# B&R Automation Studio project SD_SMA_SCADA_DEMO
Automation Studio 4.12.9.18 SP; technology packages: mapp 5.24.3, mappView 5.24.4

## Configuration Config1

CPU X20CP3687X, AutomationRuntime M4.93, Build 4.1.2, Safety 0.0, Vc V4.73.2

### Task classes (Cpu.sw)
```
Cyclic#4:
  AlarmQuerr <- AlarmQuerry.prg
  Trend <- Trend.prg
Binaries: udbdef, mvLoader, FWRules, TCData, arsvcreg, TCLang, sysconf, Role, User, iomap, ashwd, asfw, arconfig, ashwac, TC
Libraries: AsHttp, runtime, asstring, AsBrStr, sys_lib, LxVar, BrRand, MpAlarm, MpBase, arssl, fileio, astime, asieccon, brsystem, MpReport, standard
```

### Hardware
```
X20CP3687X : X20CP3687X v1.6.2.0
  Connector IF2:
    ActivateDevice = 1
    Mode = Manual
    InternetAddress = 192.168.50.233
    SubnetMask = 255.255.255.0
    InaPort = 0
    ActivateSnmp = 2
  ConfigurationID = SD_SMA_SCADA_DEMO_Config1
  UserPartitionSize = 100
  FileDevice1
  FileDeviceName1 = USER
  FileDevicePath1 = USER_PATH
  FtpUser1
  FtpUsername1 = br
  FtpUserPassword1 = JPl1VVziIj5tK4ypV/PCMk3zrwuEHr3/unO+8TvKNbo=  // 123
  FtpUserSalt1 = TmpN9Vd5
  FTPAccessRight1 = 0
  WebServerWebDir = D:\web\CFCARD\WEBROOT\
  WebServerStartPage = line.html
  ActivateOpcUa = 1
  OpcUaInformationModels_PV_Version = 1
```

## Configuration Config2

CPU X20CP3687X, AutomationRuntime M4.93, Build 4.1.2, Safety 0.0, Vc V4.73.2

### Task classes (Cpu.sw)
```
Cyclic#4:
  DataGen <- DataGen.prg
  DataRev <- DataRev.prg
  AlarmQuerr <- AlarmQuerry.prg [disabled]
  Trend <- Trend.prg [disabled]
Binaries: udbdef, mvLoader, FWRules, TCData, arsvcreg, TCLang, sysconf, Role, User, iomap, ashwd, asfw, arconfig, ashwac, TC
Libraries: AsHttp, runtime, asstring, AsBrStr, sys_lib, LxVar, BrRand, MpAlarm, MpBase, MpReport, arssl, fileio, astime, asieccon, brsystem
```

### Hardware
```
X20CP3687X : X20CP3687X v1.6.2.0
  Connector IF2:
    ActivateDevice = 1
    Mode = Manual
    InternetAddress = 192.168.50.233
    SubnetMask = 255.255.255.0
    InaPort = 0
    ActivateSnmp = 2
  ConfigurationID = SD_SMA_SCADA_DEMO_Config1
  UserPartitionSize = 100
  Simulation = 1
  FileDevice1
  FileDeviceName1 = USER
  FileDevicePath1 = USER_PATH
  FtpUser1
  FtpUsername1 = br
  FtpUserPassword1 = JPl1VVziIj5tK4ypV/PCMk3zrwuEHr3/unO+8TvKNbo=  // 123
  FtpUserSalt1 = TmpN9Vd5
  FTPAccessRight1 = 0
  WebServerWebDir = D:\web\CFCARD\WEBROOT\
  WebServerStartPage = line.html
  ActivateOpcUa = 1
  OpcUaInformationModels_PV_Version = 1
```

## Configuration PC3100

CPU X20CP1586, AutomationRuntime J4.93, Build 4.1.2, Safety 0.0, Vc V4.73.2

## Configuration cp1586

CPU 5APC3100.KBU2-000, AutomationRuntime J4.93, Build 4.1.2, Safety 0.0, Vc V4.73.2

### Task classes (Cpu.sw)
```
Cyclic#1:
  TimeSt <- TimeSt.prg
Cyclic#4:
  DataGen <- DataGen.prg
  DataRev <- DataRev.prg
  AlarmQuerr <- AlarmQuerry.prg
  Trend <- Trend.prg
  ParallelTe <- ParallelTest.prg
Binaries: udbdef, mvLoader, FWRules, TCData, arsvcreg, TCLang, sysconf, Role, User, iomap, ashwd, asfw, arconfig, ashwac, TC
Libraries: AsHttp, runtime, asstring, AsBrStr, sys_lib, LxVar, BrRand, MpAlarm, MpBase, MpReport, standard, arssl, fileio, astime, asieccon, brsystem
```

### Hardware
```
X20CP1586 : X20CP1586 v1.10.0.0
  Connector IF2:
    ActivateDevice = 1
    Mode = Manual
    InternetAddress = 192.168.50.233
    SubnetMask = 255.255.255.0
    InaPort = 0
    ActivateSnmp = 2
  Connector IF3:
    CycleTime = 400
  ConfigurationID = SD_SMA_SCADA_DEMO_Config1
  UserPartitionSize = 100
  FileDevice1
  FileDeviceName1 = USER
  FileDevicePath1 = USER_PATH
  FtpUser1
  FtpUsername1 = br
  FtpUserPassword1 = JPl1VVziIj5tK4ypV/PCMk3zrwuEHr3/unO+8TvKNbo=  // 123
  FtpUserSalt1 = TmpN9Vd5
  FTPAccessRight1 = 0
  WebServerWebDir = D:\web\CFCARD\WEBROOT\
  WebServerStartPage = line.html
  ActivateOpcUa = 1
  OpcUaInformationModels_PV_Version = 1
```

## Logical view

Binary libraries used (declarations not repeated): operator, runtime, astime, AsIecCon, AsHttp, asstring, AsBrStr, sys_lib, MpAlarm 5.24.3, MpBase, MpReport 5.24.3, standard

### Global.typ - Global data types
```iecst
TYPE
	dbReadConfig_typ : 	STRUCT
		strStartTime : ARRAY[0..DB_READ_QUERY_SIZE_MINUS_ONE]OF STRING[20];
		strEndTime : ARRAY[0..DB_READ_QUERY_SIZE_MINUS_ONE]OF STRING[20];
		strPointName : ARRAY[0..DB_READ_QUERY_SIZE_MINUS_ONE]OF STRING[20];
	END_STRUCT;
	dbReadRev_typ : 	STRUCT
		rRevBuffer : ARRAY[0..REV_BUFFER_SIZE_MINUS_ONE]OF REAL;
		udiRevTime : ARRAY[0..REV_BUFFER_SIZE_MINUS_ONE]OF UDINT;
		udiRevFeedBack : UDINT;
	END_STRUCT;
	dbReadQuery_typ : 	STRUCT
		stConfig : dbReadConfig_typ;
		stCmd : dbReadCmd_typ;
		stRev : ARRAY[0..DB_READ_QUERY_SIZE_MINUS_ONE]OF dbReadRev_typ;
	END_STRUCT;
	dbReadCmd_typ : 	STRUCT
		bNext : BOOL;
	END_STRUCT;
END_TYPE
```

### Global.var - Global variables
```iecst
VAR CONSTANT
	REV_BUFFER_SIZE : UINT := 10000;
	REV_BUFFER_SIZE_MINUS_ONE : UINT := REV_BUFFER_SIZE-1;
	DB_READ_QUERY_SIZE : UINT := 10;
	DB_READ_QUERY_SIZE_MINUS_ONE : UINT := DB_READ_QUERY_SIZE-1;
END_VAR
(*Insert your comment here.*)
VAR
	guiDBHeartBeat : UINT;
END_VAR
```

### Package Logical/Libraries - Global libraries

### Library Logical/Libraries/LxVar (ANSIC, version 1.00.4)
Depends on: AsBrStr, sys_lib

#### openErrorList.txt
```
VarHandleY:
7001:读取的变量为枚举类型
7002:DataJoint接收的指针为NULL
7003:传入DataJoint的SrcPvInfo数据丢失
7004:DataJoint拼接数据流超出设定的Buffer。
7005:DataSeperate接收的指针为NULL
7006:传入DataSeperate的SrcPvInfo数据丢失
7007:DataSeperate解析分割数据流超出设定的Buffer。
7008：JudgeSrcPvInfoNumY被传入的地址为空
7009: JudgeSrcPvInfoNumY被传入的数据所占空间为空

XmlFileY:
8001: TranGetPv2PLKPre收到的两个指针为空
8002: TranGetPv2PLKPre收到的两个长度为0
8003: TranGetPv2PLKPre在判断GetPvInfo的有效数据长度为0
8004：TranGetPv2PLKPre接收到的PLKPre数组内容超限，不能再记录更多数据，请扩展PLKPre数组长度。
8005:TranGetPv2PLKPre在转换数据流udIndex数据过大 >99999
8006:TranGetPv2PLKPre在转换数据流pStruPvInfo->sName为空
8007:TranGetPv2PLKPre在转换数据流pStruPvInfo->sDataType为空
8008:TranGetPv2PLKPre在转换数据流udLenth数据过大 >99999
8009:TranGetPv2PLKPre在转换数据流udLenth为0
8010：JudgePLKPreNum被传入的地址为空
8011: JudgePLKPreNum被传入的数据所占空间为空

8012: TranPLKPre2GetPv收到的两个指针为空
8013: TranPLKPre2GetPv收到的两个长度为0
8014: TranPLKPre2GetPv在判断PLKPre的有效数据长度为0
8015：TranPLKPre2GetPv接收到的GetPvInfo数组内容超限，不能再记录更多数据，请扩展GetPvInfo数组长度。
8016:TranPLKPre2GetPv在转换得到的数据流PLKPreDataUser.sIndex为空数据
8017:TranPLKPre2GetPv在转换得到的数据流udIndex数据过大 >99999 或过小 < 0
8018:TranPLKPre2GetPv在转换数据流pStruPreData->sName为空
8019:TranPLKPre2GetPv在转换数据流pStruPreData->sDataType为空
8020:TranPLKPre2GetPv在转换得到的数据流PLKPreDataUser.sDataLen为空数据
8021:TranPLKPre2GetPv在转换得到的数据流udDataLen数据过大 >99999 或过小 < 0
8022:TranPLKPre2GetPv在转换得到的数据流udIndex数据与实际索引不匹配

8023:PLKPreDataWrite得到的指针存在为空
8024:PLKPreDataWrite接受的到数组范围值存在为0
8025:PLKPreDataWrite接受的文件名以及设备名存在空
8026:PLKPreDataWrite收到的PLKPreData源数据有效数据长度为0
8027:PLKPreDataWrite在STEP3.1进行XML分配内存出错
8028:PLKPreDataWrite在STEP3.2进行XML文件头创建出错
8029:PLKPreDataWrite在STEP3.3进行创建头信息PLKPreData出错
8030:PLKPreDataWrite在STEP3.4.2进行元素头编写出错
8031:PLKPreDataWrite在STEP3.4.3进行元素Index属性赋值出错
8032:PLKPreDataWrite在STEP3.4.3进行元素ModuleName属性赋值出错
8033:PLKPreDataWrite在STEP3.4.3进行元素Name属性赋值出错
8034:PLKPreDataWrite在STEP3.4.3进行元素DataType属性赋值出错
8035:PLKPreDataWrite在STEP3.4.3进行元素DataLen属性赋值出错
8036:PLKPreDataWrite在STEP3.4.4进行关闭Data元素出错
8037:PLKPreDataWrite在STEP3.3.1进行关闭PLKPreData元素出错
8038:PLKPreDataWrite在STEP3.2.1进行关闭XML文档出错
8039:PLKPreDataWrite在STEP3.5进行XML文件内存信息获取出错
8040:PLKPreDataWrite在STEP4进行进行文件写操作出错

8041:PLKPreDataRead接收到的指针存在空。
8042:PLKPreDataRead接收到的值的长度范围存在空。
8043:PLKPreDataRead在STEP 2 FileInfo文件失败。
8045:PLKPreDataRead在STEP 3 FileReadY文件失败
8046:PLKPreDataRead在STEP 4.1 xmlCreateMemoryReader失败
8047:PLKPreDataRead在STEP 4.3 xmlReadNextNode失败
8048：PLKPreDataRead在STEP 4.3.2 xmlReadAttributeNr读取失败
8049：PLKPreDataRead在STEP 4.5内存读取关闭出错
8050：PLKPreDataRead在STEP 4.3.3读取的Node数据超过可容纳上限。请增大pPLKPreData对应的数组长度
8051：PLKPreDataRead在STEP4.3.0 Node真正需要的Name与Size数据空间大小过小
8052：PLKPreDataRead在STEP4.3.2.1 Attr真正需要的Name与Size数据空间大小过小
```

#### Types.typ - Exported data types
```iecst
TYPE
	GetPvInfoUser_typ : 	STRUCT
		udPvAddr : UDINT;
		sDataType : STRING[19];
		udLenth : UDINT;
		sModuleName : STRING[21];
		sName : STRING[65];
	END_STRUCT;
	DataJointUser_typ : 	STRUCT
		sCurrentName : STRING[65];
		sCurrentModName : STRING[21];
		udCurrentOffset : UDINT;
		udDataIndex : UDINT;
		udBufferMaxLen : UDINT;
		pBuffer : UDINT;
		pSrcPvInfo : UDINT;
		udSrcPvInfoNum : UDINT;
		status : UINT;
		sErrLogMessage : STRING[160];
	END_STRUCT;
	DataSeperateUser_typ : 	STRUCT
		sCurrentName : STRING[65];
		sCurrentModName : STRING[21];
		udCurrentOffset : UDINT;
		udDataIndex : UDINT;
		udBufferMaxLen : UDINT;
		pBuffer : UDINT;
		pSrcPvInfo : UDINT;
		udSrcPvInfoNum : UDINT;
		status : UINT;
		sErrLogMessage : STRING[160];
	END_STRUCT;
	JudgeSrcPvInfoNumUser_typ : 	STRUCT
		pPvArrInstance : UDINT;
		udPvArrInstanceLen : UDINT;
		udSrcNum : UDINT;
		status : UINT;
	END_STRUCT;
	LxData_Tmp_Value_typ : 	STRUCT
		bBOOL : BOOL;
		iSINT : SINT;
		iINT : INT;
		iDINT : DINT;
		uUSINT : USINT;
		uUINT : UINT;
		uUDINT : UDINT;
		rREAL : REAL;
		tDATA_AND_TIME : DATE_AND_TIME;
		tTIME : TIME;
		tDATE : DATE;
		rLREAL : LREAL;
	END_STRUCT;
END_TYPE
```

#### Constants.var - Exported constants
```iecst
VAR CONSTANT
	GET_STRU_PV_NAME_SIZE : UINT := 200; (*获取成员变量名的数组空间大小*)
	MODULE_PV_NAME_STR_SIZE : USINT := 107; (*包含 [ 任务名 : 变量名 ] 的字符串大小*)
	NAME_STR_SIZE : USINT := 65; (*包含 [ 变量名 ] 的字符串大小*)
	SHOW_LOCAL_PV_ADDR_SIZE : USINT := 80; (*显示局部变量地址实际USINT字节映射的缓存数组大小*)
END_VAR
```

#### LxVar.fun - Exported functions and function blocks
```iecst
{REDUND_ERROR} FUNCTION_BLOCK FB_GetPvInfo (*通过任务名+变量名，获得地址、数据类型、数据长度信息*) (*$GROUP=User,$CAT=User,$GROUPICON=User.png,$CATICON=User.png*)
	VAR_INPUT
		sAppModuleName : STRING[20]; (*任务名:需注意超过10个字符会自动缩写。以Cpu.sw中信息为准*)
		sName : STRING[65]; (*变量名*)
		sCompleteName : STRING[107]; (*(可选)可带任务名的完整变量名称。如果此变量有值，则sModuleName与sName不起作用。*)
	END_VAR
	VAR_OUTPUT
		udPvAddr : {REDUND_UNREPLICABLE} UDINT; (*变量地址*)
		sDataType : {REDUND_UNREPLICABLE} STRING[18]; (*字符串类型的数据类型*)
		udLenth : {REDUND_UNREPLICABLE} UDINT; (*变量实际占用长度*)
		sPvName : STRING[107]; (*内部拼接的变量名*)
		uDataType : UDINT; (*数据类型的变量类型*)
		status : UINT; (*返回状态信息，0则为正常*)
		uiDimension : UINT;
	END_VAR
	VAR
		udData_typ : UDINT;
		udData_len : UDINT;
		sDelimiter : STRING[2];
	END_VAR
END_FUNCTION_BLOCK

{REDUND_ERROR} FUNCTION GetPvOutside : UINT (*将变量信息获取并输出至外部数据结构中*) (*$GROUP=User,$CAT=User,$GROUPICON=User.png,$CATICON=User.png*)
	VAR_INPUT
		dataIn : GetPvInfoUser_typ;
	END_VAR
END_FUNCTION

{REDUND_ERROR} FUNCTION DataJoint : UINT (*根据地址，数据拼接*) (*$GROUP=User,$CAT=User,$GROUPICON=User.png,$CATICON=User.png*)
	VAR_INPUT
		DataIn : DataJointUser_typ;
	END_VAR
END_FUNCTION

{REDUND_ERROR} FUNCTION DataSeparate : UINT (*根据地址，数据拆分*) (*$GROUP=User,$CAT=User,$GROUPICON=User.png,$CATICON=User.png*)
	VAR_INPUT
		DataIn : DataSeperateUser_typ;
	END_VAR
END_FUNCTION

{REDUND_ERROR} FUNCTION JudgeSrcPvInfoNum : UINT (*判断GetPvInfoUser数组结构有效长度*) (*$GROUP=User,$CAT=User,$GROUPICON=User.png,$CATICON=User.png*)
	VAR_INPUT
		DataIn : JudgeSrcPvInfoNumUser_typ;
	END_VAR
END_FUNCTION

FUNCTION_BLOCK FB_GetModuleName (*获取调用此功能块的任务名*)
	VAR_OUTPUT
		strOut : STRING[20];
	END_VAR
	VAR
		udCheckCallCount : UDINT := 0;
	END_VAR
END_FUNCTION_BLOCK

FUNCTION_BLOCK FB_GetLocalPvAddr (*获取局部变量地址信息，可生成字符串信息并生成logger*)
	VAR_INPUT
		bWriteLogEnableFlag : BOOL := FALSE;
		sPvName : STRING[65];
	END_VAR
	VAR_OUTPUT
		udAddr : UDINT;
		strOut : STRING[130];
	END_VAR
	VAR
		udCheckCallCount : UDINT;
		FB_GetPvInfoY : FB_GetPvInfo;
		FB_GetModuleNameY : FB_GetModuleName;
		FB_Udint2StrY : FB_Udint2Str;
		sPvNameTmp : STRING[65];
	END_VAR
END_FUNCTION_BLOCK

FUNCTION_BLOCK FB_GetPvAddrStr (*获取变量地址信息，可生成字符串信息并生成logger*)
	VAR_INPUT
		bWriteLogEnableFlag : BOOL := FALSE;
		sModuleName : STRING[20];
		sPvName : STRING[65];
	END_VAR
	VAR_OUTPUT
		udAddr : UDINT;
		strOut : STRING[130];
		uStatus : UINT;
	END_VAR
	VAR
		udCheckCallCount : UDINT;
		FB_GetPvInfoY : FB_GetPvInfo;
		FB_Udint2StrY : FB_Udint2Str;
		sPvNameTmp : STRING[65];
		sModuleNameTmp : STRING[20];
	END_VAR
END_FUNCTION_BLOCK

{REDUND_ERROR} FUNCTION_BLOCK FB_GetStruPvMemName (*支持局部以及全局的变量列出其包含的成员变量名*) (*$GROUP=User,$CAT=User,$GROUPICON=User.png,$CATICON=User.png*)
	VAR_INPUT
		LocalFlag : BOOL;
		sModuleName : STRING[20];
		sName : {REDUND_UNREPLICABLE} STRING[NAME_STR_SIZE];
		sCompleteName : STRING[107]; (*(可选)可带任务名的完整变量名称。如果此变量有值，则sModuleName与sName不起作用。*)
	END_VAR
	VAR_OUTPUT
		sArrMemName : ARRAY[0..GET_STRU_PV_NAME_SIZE] OF STRING[MODULE_PV_NAME_STR_SIZE];
		uiMemNum : UINT;
		uiStatus : UINT;
	END_VAR
	VAR
		uiIndex : UINT;
		sPvName : STRING[MODULE_PV_NAME_STR_SIZE];
		udCheckCallCount : UDINT;
		sModulePvName : USINT;
		sModuleNameTmp : STRING[20];
		sNameTmp : STRING[NAME_STR_SIZE];
		FB_GetModuleNameY : FB_GetModuleName;
		sCompleteNameTmp : STRING[107];
	END_VAR
END_FUNCTION_BLOCK

{REDUND_ERROR} FUNCTION_BLOCK FB_ShowLocalPvAddrData (*显示局部变量的地址范围内内存分配*) (*$GROUP=User,$CAT=User,$GROUPICON=User.png,$CATICON=User.png*)
	VAR_INPUT
		sName : {REDUND_UNREPLICABLE} STRING[NAME_STR_SIZE];
	END_VAR
	VAR_OUTPUT
		usArrData : {REDUND_UNREPLICABLE} ARRAY[0..SHOW_LOCAL_PV_ADDR_SIZE] OF USINT;
		udAddr : UDINT;
	END_VAR
	VAR
		sNameTmp : STRING[NAME_STR_SIZE];
		FB_GetLocalPvAddrStrY : FB_GetLocalPvAddr;
		udCheckCallCount : UDINT;
	END_VAR
END_FUNCTION_BLOCK

{REDUND_ERROR} FUNCTION_BLOCK FB_ShowAddrData (*输入地址，显示地址前后一段空间的内存分布*) (*$GROUP=User,$CAT=User,$GROUPICON=User.png,$CATICON=User.png*)
	VAR_INPUT
		pWatchAddr : UDINT; (*观察数据分布的地址输入*)
		bContinuousWatch : BOOL; (*如果开启，则连续更新数据*)
		iOffset : DINT; (*对应变量地址的数据偏移，便于查看数据*)
	END_VAR
	VAR_OUTPUT
		udCurrentAddr : {REDUND_UNREPLICABLE} UDINT;
		auData : {REDUND_UNREPLICABLE} ARRAY[0..SHOW_LOCAL_PV_ADDR_SIZE] OF USINT;
		sData : STRING[SHOW_LOCAL_PV_ADDR_SIZE];
		auDataBefore : ARRAY[0..SHOW_LOCAL_PV_ADDR_SIZE] OF USINT;
		sDataBefore : STRING[SHOW_LOCAL_PV_ADDR_SIZE];
		uStatus : UINT;
	END_VAR
	VAR
		udCheckCallCount : {REDUND_UNREPLICABLE} UDINT;
		pWatchAddrTmp : UDINT;
		iOffsetTmp : DINT;
	END_VAR
END_FUNCTION_BLOCK

{REDUND_ERROR} FUNCTION_BLOCK FB_ShowPvAddrData (*显示变量的地址前后范围的实际数据*) (*$GROUP=User,$CAT=User,$GROUPICON=User.png,$CATICON=User.png*)
	VAR_INPUT
		sModuleName : {REDUND_UNREPLICABLE} STRING[20];
		sName : {REDUND_UNREPLICABLE} STRING[NAME_STR_SIZE];
		bContinuousWatch : BOOL; (*如果开启，则连续更新数据*)
		iOffset : DINT; (*对应变量地址的数据偏移，便于查看数据*)
	END_VAR
	VAR_OUTPUT
		auData : {REDUND_UNREPLICABLE} ARRAY[0..SHOW_LOCAL_PV_ADDR_SIZE] OF USINT;
		udAddr : {REDUND_UNREPLICABLE} UDINT;
		uStatus : UINT;
		sData : STRING[SHOW_LOCAL_PV_ADDR_SIZE];
		auDataBefore : ARRAY[0..SHOW_LOCAL_PV_ADDR_SIZE] OF USINT;
		sDataBefore : STRING[SHOW_LOCAL_PV_ADDR_SIZE];
	END_VAR
	VAR
		sModuleNameTmp : STRING[20];
		sNameTmp : {REDUND_UNREPLICABLE} STRING[NAME_STR_SIZE];
		FB_GetPvAddrStr_0 : {REDUND_UNREPLICABLE} FB_GetPvAddrStr;
		udCheckCallCount : {REDUND_UNREPLICABLE} UDINT;
		iOffsetTmp : DINT;
	END_VAR
END_FUNCTION_BLOCK

{REDUND_ERROR} FUNCTION Strcats : UDINT (*基于strlcat实现的缓冲区溢出保护的strcat*) (*$GROUP=User,$CAT=User,$GROUPICON=User.png,$CATICON=User.png*)
	VAR_INPUT
		pDest : UDINT;
		udDestsz : UDINT;
		pSrc : UDINT;
	END_VAR
END_FUNCTION

{REDUND_ERROR} FUNCTION Strcpys : UDINT (*基于strlcpy实现的缓冲区溢出保护的strcpy*) (*$GROUP=User,$CAT=User,$GROUPICON=User.png,$CATICON=User.png*)
	VAR_INPUT
		pDest : UDINT;
		udDestsz : UDINT;
		pSrc : UDINT;
	END_VAR
END_FUNCTION

{REDUND_ERROR} FUNCTION Strlens : UDINT (*带有最大长度限制的字符串长度统计函数*) (*$GROUP=User,$CAT=User,$GROUPICON=User.png,$CATICON=User.png*)
	VAR_INPUT
		pStr : UDINT;
		udMaxSize : UDINT;
	END_VAR
END_FUNCTION

FUNCTION_BLOCK FB_Udint2Str (*将UDINT类型数据转换为STRING*)
	VAR_INPUT
		udInput : UDINT;
	END_VAR
	VAR_OUTPUT
		strOut : STRING[14];
		uiLen : UINT;
	END_VAR
END_FUNCTION_BLOCK

{REDUND_ERROR} FUNCTION_BLOCK FB_Real2Str (*带有小数点限制的REAL数据转换*) (*$GROUP=User,$CAT=User,$GROUPICON=User.png,$CATICON=User.png*)
	VAR_INPUT
		rNum : REAL;
		digital : {REDUND_UNREPLICABLE} USINT := 2;
	END_VAR
	VAR_OUTPUT
		strOut : {REDUND_UNREPLICABLE} STRING[32];
		uiLen : UINT;
	END_VAR
END_FUNCTION_BLOCK

{REDUND_ERROR} {REDUND_UNREPLICABLE} FUNCTION_BLOCK FB_LReal2Str (*带有小数点限制的LREAL数据转换*) (*$GROUP=User,$CAT=User,$GROUPICON=User.png,$CATICON=User.png*)
	VAR_INPUT
		rNum : {REDUND_UNREPLICABLE} LREAL;
		digital : {REDUND_UNREPLICABLE} USINT := 2;
	END_VAR
	VAR_OUTPUT
		strOut : {REDUND_UNREPLICABLE} STRING[32];
		uiLen : {REDUND_UNREPLICABLE} UINT;
	END_VAR
END_FUNCTION_BLOCK

{REDUND_ERROR} FUNCTION VarWarnLogWrite : UINT (*在System中写Logger函数*) (*$GROUP=User,$CAT=User,$GROUPICON=User.png,$CATICON=User.png*)
	VAR_INPUT
		uNum : UINT;
		psErrorInfo : UDINT;
	END_VAR
END_FUNCTION

{REDUND_ERROR} {REDUND_UNREPLICABLE} FUNCTION_BLOCK FB_Dec2Hex (*十进制数据转换为十六进制字符串数据*) (*$GROUP=User,$CAT=User,$GROUPICON=User.png,$CATICON=User.png*)
	VAR_INPUT
		iDec : {REDUND_UNREPLICABLE} DINT;
	END_VAR
	VAR_OUTPUT
		sHex : {REDUND_UNREPLICABLE} STRING[20];
	END_VAR
END_FUNCTION_BLOCK

{REDUND_ERROR} FUNCTION_BLOCK FB_Hex2Dec (*十六进制字符串数据转换为十进制数据*) (*$GROUP=User,$CAT=User,$GROUPICON=User.png,$CATICON=User.png*)
	VAR_INPUT
		sHex : {REDUND_UNREPLICABLE} STRING[20];
	END_VAR
	VAR_OUTPUT
		iDec : DINT;
	END_VAR
END_FUNCTION_BLOCK

{REDUND_ERROR} FUNCTION_BLOCK FB_GetPvEntireName (*输入变量，判断是否为基本数据类型，如果不是，则返回下一级信息*) (*$GROUP=User,$CAT=User,$GROUPICON=User.png,$CATICON=User.png*)
	VAR_INPUT
		sModuleName : STRING[20]; (*任务名:需注意超过10个字符会自动缩写。以Cpu.sw中信息为准*)
		sName : STRING[65]; (*变量名*)
		sCompleteName : STRING[107]; (*(可选)可带任务名的完整变量名称。如果此变量有值，则sModuleName与sName不起作用。*)
	END_VAR
	VAR_OUTPUT
		uStatus : UINT;
		sEntirePvName : STRING[107];
		uCurrentIndex : UDINT;
		uTotalNumber : UDINT;
		bInTraversal : BOOL; (*标志位：正在遍历数组/结构体的成员*)
		bEnd : BOOL; (*代表变量不是结构体或者数组，无需再递归获取其变量名。*)
	END_VAR
	VAR
		sModuleNameTmp : STRING[20]; (*任务名:需注意超过10个字符会自动缩写。以Cpu.sw中信息为准*)
		sNameTmp : STRING[65]; (*变量名*)
		FB_GetPvInfo_0 : FB_GetPvInfo;
		FB_GetStruPvMemName_0 : FB_GetStruPvMemName;
		FB_Udint2Str_0 : FB_Udint2Str;
		sCompleteNameTmp : STRING[107];
	END_VAR
END_FUNCTION_BLOCK

{REDUND_ERROR} FUNCTION VarServLogWrite : BOOL (*在System中写Logger函数，PLC进入SERV*) (*$GROUP=User,$CAT=User,$GROUPICON=User.png,$CATICON=User.png*)
	VAR_INPUT
		uErrorNum : UINT;
		psErrorInfo : UDINT;
	END_VAR
END_FUNCTION

{REDUND_ERROR} FUNCTION ReturnPvAddr : UDINT (*可获得变量地址信息，如果找不到，则进入SERV*) (*$GROUP=User,$CAT=User,$GROUPICON=User.png,$CATICON=User.png*)
	VAR_INPUT
		psVarName : UDINT;
	END_VAR
END_FUNCTION

{REDUND_ERROR} FUNCTION_BLOCK FB_ContinualStrcat (*可具有保护的,用于连续strcat操作的函数,避免负载过高*) (*$GROUP=User,$CAT=User,$GROUPICON=User.png,$CATICON=User.png*)
	VAR_INPUT
		psDestStr : {REDUND_UNREPLICABLE} UDINT;
		uDestMaxSize : {REDUND_UNREPLICABLE} UDINT; (*[ 可选 ] 若不输入，则不进行安全检查*)
		psSrcStr : {REDUND_UNREPLICABLE} UDINT;
		uSrcMaxSize : {REDUND_UNREPLICABLE} UDINT; (*[ 可选 ] 若不输入，则不进行安全检查*)
		bInitial : BOOL; (*若为TRUE，则uOffset归0，第一次调用此功能块的时候需使用*)
		uDestStrOffset : UDINT; (*[ 可选 ] 目标字符串的某一偏移量开始进行字符串添加，不影响功能，可用于降低strcat负载*)
	END_VAR
	VAR_OUTPUT
		uStrSize : UDINT;
		uStatus : {REDUND_UNREPLICABLE} UINT;
	END_VAR
	VAR
		uOffset : {REDUND_UNREPLICABLE} UDINT;
		uSrcActualLenth : UDINT;
		uDestInitialLenth : UDINT;
	END_VAR
END_FUNCTION_BLOCK
```

#### FB_GetPvInfo.c - 获取变量的地址、长度、类型等信息
```c
/*!
	* @file       FB_GetPvInfo.c
	* @brief      调用此函数，可获得任何变量的地址、数据类型、数据长度等信息。
	* @date       创建于：2018.02.19；最后修改日期：2021.06.03
	* @version    V 1.00.5
	* @author     YuanZhiyi
	* @copyright  B&R
*/
/*! History
 *****************************************************************************
 *     2018.02.19    V1.00.1   YuanZhiyi
 *         (new)     初始版本
 *     2021.03.05    V1.00.2   YuanZhiyi
 *         (fix)     调整代码的_LOCAL写法，避免在部分AS中编译异常问题。
 *     2021.03.15    V1.00.3   YuanZhiyi
 *         (fix)     调整uiDimension变量方向为VAR_OUTPUT,并修正此参数的数据长度。
 *     2021.03.16    V1.00.4   YuanZhiyi
 *         (new)     增加sCompleteName，满足后续输出内容直接获取地址。
 *     2021.06.03    V1.00.5   YuanZhiyi
 *         (fix)     修正当数据为枚举类型或结构体时，无法获得地址的设计
 ******************************************************************************
*/

#include <bur/plctypes.h>
#ifdef __cplusplus
	extern "C"
	{
#endif
	#include "LxVar.h"
	#include <sys_lib.h>
	#include <string.h>
#ifdef __cplusplus
	};
#endif

void FB_GetPvInfo(struct FB_GetPvInfo* inst)
{
	//注意事项：	不进行步骤跳转，一个任务周期内即完成所有任务
	//STEP 0: 初始化

	memcpy((char *)inst->sDelimiter, (char *)":",1);

	memset((char *)&inst->udPvAddr, 0, 4);
	memset((char *)inst->sDataType, 0, 19);
	memset((char *)&inst->udLenth, 0, 4);
	memset((char *)&inst->udData_typ, 0, 4);
	memset((char *)&inst->udData_len, 0, 4);
	memset((char *)&inst->uiDimension, 0, 1);

	//STEP 1: 判断输入数据是否正常
	memset((char *)inst->sPvName, 0, sizeof(inst->sPvName)); //清空缓存
    if (memcmp((char *)inst->sCompleteName,(char *)"",1) != 0) { //判断是否启用sCompleteName:使用sCompleteName
        memcpy((char *)inst->sPvName, (char *)inst->sCompleteName,sizeof(inst->sCompleteName));
        memset((char *)inst->sAppModuleName,0,sizeof(inst->sAppModuleName));
        memset((char *)inst->sName,0,sizeof(inst->sName));
    }else { //使用sAppModuleName与sName
	    if (memcmp((char *)inst->sAppModuleName,(char *)"",1) == 0){
		    strcat((char *)inst->sPvName,(char *)inst->sName);
	    }else{
		    strcat((char *)inst->sPvName,(char *)inst->sAppModuleName);
		    strcat((char *)inst->sPvName,(char *)inst->sDelimiter);
		    strcat((char *)inst->sPvName,(char *)inst->sName);
	    }
    }
	//STEP 2: 进行PV_ninfo，判断数据类型，是否返回错误数据
	inst->status = PV_ninfo((char *)inst->sPvName, (UDINT *)&inst->udData_typ, (UDINT *)&inst->udData_len, (UINT *)&inst->uiDimension);
	//因上一语句处理完，则inst->sPvName的值会被清空，因而做了以下操作
	memset((char *)inst->sPvName, 0, sizeof(inst->sPvName)); //清空缓存
    if (memcmp((char *)inst->sCompleteName,(char *)"",1) != 0) { //判断是否启用sCompleteName:使用sCompleteName
        memcpy((char *)inst->sPvName, (char *)inst->sCompleteName,sizeof(inst->sCompleteName));
    }else { //任务名 变量名 分开输入
        if (memcmp((char *)inst->sAppModuleName,(char *)"",1) == 0){
            strcat((char *)inst->sPvName,(char *)inst->sName);
        }else{
            strcat((char *)inst->sPvName,(char *)inst->sAppModuleName);
            memcpy((char *)inst->sDelimiter, (char *)":",1);
            strcat((char *)inst->sPvName,(char *)inst->sDelimiter);
            strcat((char *)inst->sPvName,(char *)inst->sName);
        }
    }
	if (inst->status == 0){
    inst->uDataType = inst->udData_typ;
		switch (inst->udData_typ){
			case 0:
				strcat((char *)inst->sDataType,(char *)"Derived data types");
				inst->status = 7001;//读取的变量为枚举类型
				break;
			case 1:
				strcat((char *)inst->sDataType,(char *)"BOOL");
				break;
			case 2:
				strcat((char *)inst->sDataType,(char *)"SINT");
				break;
			case 3:
				strcat((char *)inst->sDataType,(char *)"INT");
				break;
			case 4:
				strcat((char *)inst->sDataType,(char *)"DINT");
				break;
			case 5:
				strcat((char *)inst->sDataType,(char *)"USINT");
				break;
			case 6:
				strcat((char *)inst->sDataType,(char *)"UINT");
				break;
			case 7:
				strcat((char *)inst->sDataType,(char *)"UDINT");
				break;
			case 8:
				strcat((char *)inst->sDataType,(char *)"REAL");
				break;
			case 9:
				strcat((char *)inst->sDataType,(char *)"STRING");
				break;
			case 10:
				strcat((char *)inst->sDataType,(char *)"ULINT");
				break;
			case 11:
				strcat((char *)inst->sDataType,(char *)"DATE_AND_TIME");
				break;
			case 12:
				strcat((char *)inst->sDataType,(char *)"TIME");
				break;
			case 13:
				strcat((char *)inst->sDataType,(char *)"DATE");
				break;
			case 14:
				strcat((char *)inst->sDataType,(char *)"LREAL");
				break;
			case 15:
				strcat((char *)inst->sDataType,(char *)"Derived data types");
				inst->status = 7001;//读取的变量为枚举类型
				break;
			case 16:
				strcat((char *)inst->sDataType,(char *)"TIME_OF_DAY");
				break;
			case 17:
				strcat((char *)inst->sDataType,(char *)"BYTE");
				break;
			case 18:
				strcat((char *)inst->sDataType,(char *)"WORD");
				break;
			case 19:
				strcat((char *)inst->sDataType,(char *)"DWORD");
				break;
			case 20:
				strcat((char *)inst->sDataType,(char *)"LWORD");
				break;
			case 21:
				strcat((char *)inst->sDataType,(char *)"WSTRING");
				break;
			case 23:
				strcat((char *)inst->sDataType,(char *)"LINT");
				break;
			default:
				break;
		}
	}
	//STEP3 : 上面都通过，则进行PV_xgetadr，获取地址数据
	if (inst->status == 0 || inst->status == 7001){
		inst->status = PV_xgetadr(inst->sPvName, &inst->udPvAddr, &inst->udLenth);
	}
}
```

#### GetPvOutside.c - 将变量信息获取并输出至外部数据结构中
```c
/*!
	* @file       GetPvOutside.c
	* @brief      将变量信息获取并输出至外部数据结构中
	* @date       创建于：2018.02.19；最后修改日期：2018.02.19
	* @version    V 1.00.1
	* @author     YuanZhiyi
	* @copyright  B&R
*/
/*! History
 *****************************************************************************
 *     2018.02.19    V1.00.1   YuanZhiyi
 *         (new)     初始版本
 ******************************************************************************
*/

#include <bur/plctypes.h>
#ifdef __cplusplus
	extern "C"
	{
#endif
	#include "LxVar.h"
	#include <string.h>
#ifdef __cplusplus
	};
#endif

FB_GetPvInfo_typ GetPvInfoY_0;

unsigned short GetPvOutside(struct GetPvInfoUser_typ* dataIn)
{

	//是否增加dataIn的数据校验？
	//如果数据不正常，应该会在编译时就报错。但需要确认数据是否正常
	memcpy((char *)&GetPvInfoY_0.sAppModuleName,(char *)dataIn->sModuleName,sizeof(dataIn->sModuleName));
	memcpy((char *)GetPvInfoY_0.sName,(char *)dataIn->sName,sizeof(dataIn->sName));
	FB_GetPvInfo(&GetPvInfoY_0);
	if(GetPvInfoY_0.status == 0){
		memcpy((char *)dataIn->sDataType,(char *)GetPvInfoY_0.sDataType,19);
		dataIn->udLenth = GetPvInfoY_0.udLenth;
		dataIn->udPvAddr = GetPvInfoY_0.udPvAddr;
	}else{
		memset((char *)dataIn->sDataType,0,19);
		dataIn->udLenth = 0;
		dataIn->udPvAddr = 0;
	}
	return GetPvInfoY_0.status;
}
```

#### DataJoint.c - 根据地址，数据拼接
```c
/*!
	* @file       DataJoint.c
	* @brief      根据地址信息，实现数据拼接
	* @date       创建于：2018.02.19；最后修改日期：2018.02.19
	* @version    V 1.00.1
	* @author     YuanZhiyi
	* @copyright  B&R
*/
/*! History
 *****************************************************************************
 *     2018.02.19    V1.00.1   YuanZhiyi
 *         (new)     初始版本
 ******************************************************************************
*/

#include <bur/plctypes.h>
#ifdef __cplusplus
	extern "C"
	{
#endif
	#include "LxVar.h"
	#include <string.h>
#ifdef __cplusplus
	};
#endif

GetPvInfoUser_typ *pStruPvInfo;

unsigned short DataJoint(struct DataJointUser_typ* DataIn)
{
	//一个任务周期就需要全部完成所有任务
	//STEP 0 清空|初始化
	memset((char *)DataIn->sCurrentName,0,sizeof(DataIn->sCurrentName));
	memset((char *)DataIn->sCurrentModName,0,sizeof(DataIn->sCurrentModName));
	memset((char *)DataIn->sErrLogMessage,0,sizeof(DataIn->sErrLogMessage));
	DataIn->udCurrentOffset = 0;
	DataIn->udDataIndex = 0;
	//STEP 1 检查输入的指针是否正常
	if (DataIn->pBuffer == 0 || DataIn->pSrcPvInfo == 0){
		DataIn->status = 7002;
		return 7002; //7002:DataJoint接收的指针为NULL
	}
	//STEP 2 进入循环进行处理
	for (DataIn->udDataIndex = 0; DataIn->udDataIndex < DataIn->udSrcPvInfoNum; DataIn->udDataIndex++){
		//STEP 2.1 进行数据准备 记录当前信息
		pStruPvInfo = (GetPvInfoUser_typ *)(DataIn->pSrcPvInfo + DataIn->udDataIndex * sizeof(GetPvInfoUser_typ));
		memcpy((char *)DataIn->sCurrentName,(char *)pStruPvInfo->sName,sizeof(pStruPvInfo->sName));
		memcpy((char *)DataIn->sCurrentModName,(char *)pStruPvInfo->sModuleName,sizeof(pStruPvInfo->sModuleName));
		//STEP 2.2 检测pStruPvInfo的信息是否完整。
		if (pStruPvInfo->udPvAddr == 0 || pStruPvInfo->udLenth == 0){
			//STEP 2.2.1 当数据异常时，则将卡主的地方变量传递至sErrLogMessage，便于找到错误点。
			strcpy((char *)DataIn->sErrLogMessage,(char *)"DataJointY::PV NOT FOUND:");//sErrLogMessage总长度不能超过160字节。
			strcat((char *)DataIn->sErrLogMessage,(char *)pStruPvInfo->sName);
			DataIn->status = 7003;
			return 7003;//7003:传入DataJoint的SrcPvInfo数据丢失，即传入的数据为错误的。
		}
		//STEP 2.3 进行Buffer边界判断，是否超界。
		if (DataIn->udCurrentOffset + pStruPvInfo->udLenth > DataIn->udBufferMaxLen ){
			DataIn->status = 7004;
			return 7004;//7004:DataJoint拼接数据流超出设定的Buffer。
		}
		//STEP 2.4 进行数据复制，存储信息
		memcpy((char *)(DataIn->pBuffer + DataIn->udCurrentOffset),(char *)pStruPvInfo->udPvAddr,(UDINT)pStruPvInfo->udLenth);
		DataIn->udCurrentOffset += pStruPvInfo->udLenth;
		//break;
	}
	DataIn->status = 0;
    return 0;
}
```

#### DataSeparate.c - 根据地址，数据拆分
```c
/*!
	* @file       DataJoint.c
	* @brief      根据地址信息，实现数据拆分
	* @date       创建于：2018.02.19；最后修改日期：2018.02.19
	* @version    V 1.00.1
	* @author     YuanZhiyi
	* @copyright  B&R
*/
/*! History
 *****************************************************************************
 *     2018.02.19    V1.00.1   YuanZhiyi
 *         (new)     初始版本
 ******************************************************************************
*/

#include <bur/plctypes.h>
#ifdef __cplusplus
	extern "C"
	{
#endif
	#include "LxVar.h"
	#include <string.h>
#ifdef __cplusplus
	};
#endif

GetPvInfoUser_typ *pStruPvInfo;

unsigned short DataSeparate(struct DataSeperateUser_typ* DataIn)
{
	//一个任务周期就需要全部完成所有任务
	//STEP 0 清空|初始化
	memset((char *)DataIn->sCurrentName,0,sizeof(DataIn->sCurrentName));
	memset((char *)DataIn->sCurrentModName,0,sizeof(DataIn->sCurrentModName));
	memset((char *)DataIn->sErrLogMessage,0,sizeof(DataIn->sErrLogMessage));
	DataIn->udCurrentOffset = 0;
	DataIn->udDataIndex = 0;
	//STEP 1 检查输入的指针是否正常
	if (DataIn->pBuffer == 0 || DataIn->pSrcPvInfo == 0){
		DataIn->status = 7005;
		return 7005; //7005:DataSeperate接收的指针为NULL
	}
	//STEP 2 进入循环进行处理
	for (DataIn->udDataIndex = 0; DataIn->udDataIndex < DataIn->udSrcPvInfoNum; DataIn->udDataIndex++){	//DataIn->udSrcPvInfoNum值输入比较特殊，需要确定
		//STEP 2.1 进行数据准备 记录当前信息
		pStruPvInfo = (GetPvInfoUser_typ *)(DataIn->pSrcPvInfo + DataIn->udDataIndex * sizeof(GetPvInfoUser_typ));
		memcpy((char *)DataIn->sCurrentName,(char *)pStruPvInfo->sName,sizeof(pStruPvInfo->sName));
		memcpy((char *)DataIn->sCurrentModName,(char *)pStruPvInfo->sModuleName,sizeof(pStruPvInfo->sModuleName));
		//STEP 2.2 检测pStruPvInfo的信息是否完整。
		if (pStruPvInfo->udPvAddr == 0 || pStruPvInfo->udLenth == 0){
			//STEP 2.2.1 当数据异常时，则将卡主的地方变量传递至sErrNameSite，便于找到错误点。
			strcpy((char *)DataIn->sErrLogMessage,(char *)"DataSeparate::PV NOT FOUND:");//sErrLogMessage总长度不能超过80字节。
			strcat((char *)DataIn->sErrLogMessage,(char *)pStruPvInfo->sName);
			DataIn->status = 7006;
			return 7006;//7006:传入DataSeperate的SrcPvInfo数据丢失，即可能为错误不存在的变量。
		}
		//STEP 2.3 进行Buffer边界判断，是否超界。
		if (DataIn->udCurrentOffset + pStruPvInfo->udLenth > DataIn->udBufferMaxLen ){ //DataIn->udBufferMaxLen的值一般为SIZEOF(输入的地址)
			DataIn->status = 7007;
			return 7007;//7007:DataSeperate解析分割数据流超出设定的Buffer。
		}
		//STEP 2.4 进行数据复制，存储信息
		memcpy((char *)pStruPvInfo->udPvAddr,(char *)(DataIn->pBuffer + DataIn->udCurrentOffset),(UDINT)pStruPvInfo->udLenth);
		DataIn->udCurrentOffset += pStruPvInfo->udLenth;
		//break;
	}
	DataIn->status = 0;
    return 0;
}
```

#### JudgeSrcPvInfoNum.c - 判断GetPvInfoUser数组结构有效长度
```c
/*!
* @file        JudgeSrcPvInfoNum.c
* @brief       判断GetPvInfoUser数组结构有效长度
* @date        创建于：2018.02.19；最后修改日期：2021.06.03
* @version     V1.00.2
* @author      YuanZhiyi
* @copyright   B&R
*/
/*! History
 *****************************************************************************
 *     2018.02.19    V1.00.1   YuanZhiyi
 *         (new)     初步实现
 *     2021.06.03    V1.00.2   YuanZhiyi
 *         (new)     补充注释
 ******************************************************************************
*/

#include <bur/plctypes.h>
#ifdef __cplusplus
	extern "C"
	{
#endif
	#include "LxVar.h"
	#include <string.h>
#ifdef __cplusplus
	};
#endif

#ifndef _LOCAL
#define _LOCAL
#endif

#define DATA_TYP GetPvInfoUser_typ

DATA_TYP *pStruPvInfo;

unsigned short JudgeSrcPvInfoNum(struct JudgeSrcPvInfoNumUser_typ* DataIn)
{
	//STEP 0:判断当前输入的信息是否有效
	if (DataIn->pPvArrInstance == 0) {
		DataIn->status = 7008;
		return 7008;//7008：JudgeSrcPvInfoNumY被传入的地址为空
	}
	if (DataIn->udPvArrInstanceLen == 0) {
		DataIn->status = 7009;
		return 7009;//7009: JudgeSrcPvInfoNumY被传入的数据所占空间为空
	}
	//STEP 1:进行For循环处理，扫描判断此输入数组的数据是否足够
	for (DataIn->udSrcNum = 0; DataIn->udSrcNum < DataIn->udPvArrInstanceLen; DataIn->udSrcNum++) {
		pStruPvInfo = (DATA_TYP *)(DataIn->pPvArrInstance + DataIn->udSrcNum * sizeof(DATA_TYP));
		if (memcmp((char *)pStruPvInfo->sName,(char *)"",1) == 0) {
			DataIn->status = 0;
			return 0;
		}
	}
	DataIn->status = 0;
	return 0;
}
```

#### FB_GetModuleName.c - 获取调用此功能块的任务名
```c
/*!
	* @file        FB_GetModuleName.c
	* @brief       调用此函数，获取调用此功能块的任务名
	* @date        创建于：2019.08.13；最后修改日期：2019.08.13
	* @version     V 1.00.1
	* @author      YuanZhiyi
	* @copyright   B&R
*/
/*! History
 *****************************************************************************
 *     2019.08.13    V1.00.1   YuanZhiyi
 *         (new)     初始版本
 ******************************************************************************
*/

#include <bur/plctypes.h>
#ifdef __cplusplus
	extern "C"
	{
#endif
	#include "LxVar.h"
	#include <string.h>
	#include <sys_lib.h>
#ifdef __cplusplus
	};
#endif

void FB_GetModuleName(struct FB_GetModuleName* inst)
{
	if (inst->udCheckCallCount <= 2)
	{
			memset((char *)inst->strOut,0,sizeof(inst->strOut));
			ST_name((UDINT)0,(char *)inst->strOut,(USINT *)0);
			inst->udCheckCallCount++;
	}
}
```

#### FB_GetLocalPvAddr.c - 获取局部变量地址信息，可生成字符串信息并生成logger
```c
/*!
	* @file        FB_GetLocalPvAddr.c
	* @brief       调用此函数，输入当前模块的局部变量，无需输入模块名，即可通过srtOut得到完整的地址信息，并支持生成Logger记录信息
				   同名模块同名变量只执行一次。
	* @date        创建于：2019.08.13；最后修改日期：2019.08.13
	* @version     V 1.00.1
	* @author      YuanZhiyi
	* @copyright   B&R
*/
/*! History
 *****************************************************************************
 *     2019.08.13    V1.00.1   YuanZhiyi
 *         (new)     初始版本
 ******************************************************************************
*/

#include <bur/plctypes.h>
#ifdef __cplusplus
	extern "C"
	{
#endif
	#include "LxVar.h"
	#include <string.h>
	#include <sys_lib.h>
#ifdef __cplusplus
	};
#endif

void FB_GetLocalPvAddr(struct FB_GetLocalPvAddr* inst)
{
	//保证此函数可在被连续调用重复使用。
	if (memcmp((char *)inst->sPvName,(char *)inst->sPvNameTmp,sizeof(inst->sPvName)) != 0)
	{
		memcpy((char *)inst->sPvNameTmp,(char *)inst->sPvName,sizeof(inst->sPvName));
		inst->udCheckCallCount = 0;
	}

	if (inst->udCheckCallCount < 1)
	{
			memset((char *)inst->strOut,0,sizeof(inst->strOut));
			inst->udCheckCallCount++;
			//获取本地任务名
			FB_GetModuleName(&inst->FB_GetModuleNameY);

			//获取地址信息以及其他
			memcpy((char *)inst->FB_GetPvInfoY.sAppModuleName,(char *)inst->FB_GetModuleNameY.strOut,sizeof(inst->FB_GetModuleNameY.strOut));
			memcpy((char *)inst->FB_GetPvInfoY.sName,(char *)inst->sPvName,sizeof(inst->sPvName));
			FB_GetPvInfo(&inst->FB_GetPvInfoY);

			//输出UDINT类型的地址信息
			inst->udAddr = inst->FB_GetPvInfoY.udPvAddr;

			//进行字符串拼接
			inst->FB_Udint2StrY.udInput = inst->FB_GetPvInfoY.udPvAddr;
			FB_Udint2Str(&inst->FB_Udint2StrY);
			strcat((char *)inst->strOut,(char *)inst->FB_GetPvInfoY.sPvName);
			strcat((char *)inst->strOut,(char *)" | Addr:");
			if (inst->udAddr == 0)//判断是否读取的变量不存在
			{
				strcat((char *)inst->strOut,(char *)"PvNotExist");
			}else
			{
				strcat((char *)inst->strOut,(char *)inst->FB_Udint2StrY.strOut);
			}

			//判断是否需要写Logger信息
			if (inst->bWriteLogEnableFlag ==  1 && inst->udCheckCallCount <= 1)
			{
				VarWarnLogWrite(7200,(UDINT)inst->strOut);
			}
	}
}
```

#### FB_GetPvAddrStr.c - 获取变量地址信息，可生成字符串信息并生成logger
```c
/*!
	* @file        FB_GetPvAddrStr.c
	* @brief       调用此函数，可输入全局变量，可输入指定模块的局部变量，通过srtOut得到完整的地址信息，并支持生成Logger记录信息
				   同名模块同名变量只执行一次。
	* @date        创建于：2019.08.13；最后修改日期：2019.08.13
	* @version     V 1.00.1
	* @author      YuanZhiyi
	* @copyright   B&R
*/
/*! History
 *****************************************************************************
 *     2019.08.13    V1.00.1   YuanZhiyi
 *         (new)     初始版本
 ******************************************************************************
*/

#include <bur/plctypes.h>

#ifdef __cplusplus
	extern "C"
	{
#endif
	#include "LxVar.h"
	#include <string.h>
	#include <sys_lib.h>
#ifdef __cplusplus
	};
#endif

void FB_GetPvAddrStr(struct FB_GetPvAddrStr* inst)
{
	//保证此函数可在被连续调用重复使用。
	if ((memcmp((char *)inst->sPvName,(char *)inst->sPvNameTmp,sizeof(inst->sPvName)) != 0) ||
		(memcmp((char *)inst->sModuleName,(char *)inst->sModuleNameTmp,sizeof(inst->sModuleName)) != 0))
	{
		memcpy((char *)inst->sPvNameTmp,(char *)inst->sPvName,sizeof(inst->sPvName));
		memcpy((char *)inst->sModuleNameTmp,(char *)inst->sModuleName,sizeof(inst->sModuleName));
		inst->udCheckCallCount = 0;
	}

	if (inst->udCheckCallCount < 1)
	{
			memset((char *)inst->strOut,0,sizeof(inst->strOut));
			inst->udCheckCallCount++;

			//获取地址信息以及其他
			memcpy((char *)inst->FB_GetPvInfoY.sAppModuleName,(char *)inst->sModuleName,sizeof(inst->sModuleName));
			memcpy((char *)inst->FB_GetPvInfoY.sName,(char *)inst->sPvName,sizeof(inst->sPvName));
			FB_GetPvInfo(&inst->FB_GetPvInfoY);
      inst->uStatus = inst->FB_GetPvInfoY.status;

			//输出UDINT类型的地址信息
			inst->udAddr = inst->FB_GetPvInfoY.udPvAddr;

			//进行字符串拼接
			inst->FB_Udint2StrY.udInput = inst->FB_GetPvInfoY.udPvAddr;
			FB_Udint2Str(&inst->FB_Udint2StrY);
			strcat((char *)inst->strOut,(char *)inst->FB_GetPvInfoY.sPvName);
			strcat((char *)inst->strOut,(char *)" | Addr:");
			if (inst->udAddr == 0)//判断是否读取的变量不存在
			{
				strcat((char *)inst->strOut,(char *)" PvNotFound");
			}else
			{
				strcat((char *)inst->strOut,(char *)inst->FB_Udint2StrY.strOut);
			}
			//判断是否需要写Logger信息
			if (inst->bWriteLogEnableFlag ==  1 && inst->udCheckCallCount <= 1)
			{
				//WarnLogWriteY(7201,(UDINT)inst->strOut);
			}
	}
}
```

#### FB_GetStruPvMemName.c - 支持局部以及全局的变量列出其包含的成员变量名
```c
/*!
	* @file        FB_GetStruPvMemName.c
	* @brief       支持局部以及全局的变量列出其包含的成员变量名
	* @date        创建于：2019.08.13；最后修改日期：2019.08.13
	* @version     V 1.00.1
	* @author      YuanZhiyi
	* @copyright   B&R
*/
/*! History
 *****************************************************************************
 *     2019.08.13    V1.00.1   YuanZhiyi
 *         (new)     初始版本
 ******************************************************************************
*/

#include <bur/plctypes.h>
#include <string.h>
#include <sys_lib.h>
#ifdef __cplusplus
	extern "C"
	{
#endif
	#include "LxVar.h"
#ifdef __cplusplus
	};
#endif

void FB_GetStruPvMemName(struct FB_GetStruPvMemName* inst)
{
	//保证此函数可在被连续调用重复使用。
	if ((memcmp((char *)inst->sName,(char *)inst->sNameTmp,sizeof(inst->sName)) != 0) ||
		 (memcmp((char *)inst->sModuleName,(char *)inst->sModuleNameTmp,sizeof(inst->sModuleName)) != 0))
	{
		memcpy((char *)inst->sNameTmp,(char *)inst->sName,sizeof(inst->sName));
		if (inst->LocalFlag == 0)
		{
	 		memcpy((char *)inst->sModuleNameTmp,(char *)inst->sModuleName,sizeof(inst->sModuleName));
		}else
		{
			FB_GetModuleName(&inst->FB_GetModuleNameY);
			memcpy((char *)inst->sModuleName,(char *)inst->FB_GetModuleNameY.strOut,sizeof(inst->sModuleName));
			memcpy((char *)inst->sModuleNameTmp,(char *)inst->sModuleName,sizeof(inst->sModuleName));
		}

        memset((char *)inst->sCompleteName,0,sizeof(inst->sCompleteName));
        memset((char *)inst->sCompleteNameTmp,0,sizeof(inst->sCompleteNameTmp));
		memset((char *)inst->sPvName,0,sizeof(inst->sPvName));
		Strcats((UDINT)inst->sPvName,sizeof(inst->sPvName),(UDINT)inst->sModuleName);
		Strcats((UDINT)inst->sPvName,sizeof(inst->sPvName),(UDINT)":");
		Strcats((UDINT)inst->sPvName,sizeof(inst->sPvName),(UDINT)inst->sName);

		inst->udCheckCallCount = 0;
		inst->uiMemNum = 0;
		inst->uiStatus = 0;
	}

    //如果输入的是变量全名
    if (memcmp((char *)inst->sCompleteName,(char *)inst->sCompleteNameTmp,sizeof(inst->sCompleteNameTmp)) != 0) {
        memcpy((char *)inst->sCompleteNameTmp,(char *)inst->sCompleteName,sizeof(inst->sCompleteName));

        memset((char *)inst->sName,0,sizeof(inst->sName));
        memset((char *)inst->sNameTmp,0,sizeof(inst->sNameTmp));
        memset((char *)inst->sModuleName,0,sizeof(inst->sModuleName));
        memset((char *)inst->sModuleNameTmp,0,sizeof(inst->sModuleNameTmp));

        memcpy((char *)inst->sPvName,(char *)inst->sCompleteName,sizeof(inst->sCompleteName));

        inst->udCheckCallCount = 0;
        inst->uiMemNum = 0;
        inst->uiStatus = 0;
    }

	if (inst->udCheckCallCount < 1)
	{
		inst->udCheckCallCount++;
		memset(inst->sArrMemName,0,sizeof(inst->sArrMemName));
		for (inst->uiIndex = 0; inst->uiIndex < GET_STRU_PV_NAME_SIZE; inst->uiIndex ++)
		{
			inst->uiStatus = PV_item((char *)inst->sPvName, (UINT)inst->uiIndex, (char *)inst->sArrMemName[inst->uiIndex]);
			if (inst->uiStatus != 0)
			{
				if (inst->uiStatus == 14704)
				{
					inst->uiStatus = 0;//如果为空变量，则可认为成员列表的列出已完成
				}
                if (inst->uiStatus == 14713)
                {
                    inst->uiStatus = 0;//ERR_PV_NODETAIL,访问的是一个实际变量，并非是结构体以及数组。
                }
				return;
			}
			inst->uiMemNum = inst->uiIndex + 1;
		}
	}
}
```

#### FB_ShowPvAddrData.c - 显示变量的地址前后范围的实际数据
```c
/*!
	* @file        FB_ShowPvAddrData.c
	* @brief       显示变量的地址前后范围的实际数据
	* @date        创建于：2019.08.13；最后修改日期：2019.08.13
	* @version     V 1.00.1
	* @author      YuanZhiyi
	* @copyright   B&R
*/
/*! History
 *****************************************************************************
 *     2019.08.13    V1.00.1   YuanZhiyi
 *         (new)     初始版本
 ******************************************************************************
*/

#include <bur/plctypes.h>
#include <string.h>
#ifdef __cplusplus
	extern "C"
	{
#endif
	#include "LxVar.h"
#ifdef __cplusplus
	};
#endif

void FB_ShowPvAddrData(struct FB_ShowPvAddrData* inst)
{
    //保证此函数可在被连续调用重复使用。
    if ((memcmp((char *)inst->sName,(char *)inst->sNameTmp,sizeof(inst->sName)) != 0) ||
       (memcmp((char *)inst->sModuleName,(char *)inst->sModuleNameTmp,sizeof(inst->sModuleName)) != 0) ||
        inst->iOffset != inst->iOffsetTmp)
    {
        memcpy((char *)inst->sNameTmp,(char *)inst->sName,sizeof(inst->sName));
        memcpy((char *)inst->sModuleNameTmp,(char *)inst->sModuleName,sizeof(inst->sModuleName));
        inst->iOffsetTmp = inst->iOffset;

        inst->uStatus = 0;
        inst->udCheckCallCount = 0;
    }

    if (inst->udCheckCallCount < 1 || inst->bContinuousWatch == 1)
    {
        inst->udCheckCallCount = 1;
        memset((char *)inst->auData,0,sizeof(inst->auData));
        memset((char *)inst->sData,0,sizeof(inst->sData));
        memset((char *)inst->auDataBefore,0,sizeof(inst->auDataBefore));
        memset((char *)inst->sDataBefore,0,sizeof(inst->sDataBefore));
        memcpy((char *)inst->FB_GetPvAddrStr_0.sModuleName,(char *)inst->sModuleName,sizeof(inst->sModuleName));
        memcpy((char *)inst->FB_GetPvAddrStr_0.sPvName,(char *)inst->sName,sizeof(inst->sName));
        FB_GetPvAddrStr(&inst->FB_GetPvAddrStr_0);
        if (inst->FB_GetPvAddrStr_0.uStatus == 0 )
        {
            if (inst->FB_GetPvAddrStr_0.udAddr != 0 && (inst->FB_GetPvAddrStr_0.udAddr + inst->iOffset > SHOW_LOCAL_PV_ADDR_SIZE))
            {
                memcpy((char *)inst->auData,(char *)inst->FB_GetPvAddrStr_0.udAddr + inst->iOffset,sizeof(inst->auData));
                memcpy((char *)inst->sData,(char *)inst->FB_GetPvAddrStr_0.udAddr + inst->iOffset,sizeof(inst->sData));
                memcpy((char *)inst->auDataBefore,(char *)inst->FB_GetPvAddrStr_0.udAddr + inst->iOffset - SHOW_LOCAL_PV_ADDR_SIZE - 1,sizeof(inst->auDataBefore));
                memcpy((char *)inst->sDataBefore,(char *)inst->FB_GetPvAddrStr_0.udAddr + inst->iOffset - SHOW_LOCAL_PV_ADDR_SIZE - 1,sizeof(inst->sDataBefore));
            }else
            {
                inst->uStatus = 1;//访问得到的地址为0
            }
            inst->udAddr = inst->FB_GetPvAddrStr_0.udAddr;
        }else
        {
            inst->uStatus = inst->FB_GetPvAddrStr_0.uStatus;
        }
    }
}
```

#### FB_ShowAddrData.c - 输入地址，显示地址前后一段空间的内存分布
```c
/*!
	* @file      FB_ShowAddrData.c
	* @brief     调用此函数，可观察地址附近的内存分布情况
	* @date      创建于：2021.03.12；最后修改日期：2021.03.12
	* @version   V 1.00.1
	* @author    YuanZhiyi
	* @copyright B&R
*/
/*! History
 *****************************************************************************
 *     2021.03.12    V1.00.1   YuanZhiyi
 *         (new)     初始版本
 ******************************************************************************
*/

#include <bur/plctypes.h>
#include <string.h>
#ifdef __cplusplus
	extern "C"
	{
#endif
	#include "LxVar.h"
#ifdef __cplusplus
	};
#endif

void FB_ShowAddrData(struct FB_ShowAddrData* inst)
{
    //保证此函数可在被连续调用重复使用。
    if ((inst->pWatchAddr != inst->pWatchAddrTmp) || (inst->iOffset != inst->iOffsetTmp))
    {
        inst->pWatchAddrTmp = inst->pWatchAddr;
        inst->iOffsetTmp    = inst->iOffset;

        inst->uStatus = 0;
        inst->udCheckCallCount = 0;
    }

    if (inst->udCheckCallCount < 1 || inst->bContinuousWatch == 1)
    {
        inst->udCheckCallCount = 1;
        memset((char *)inst->auData,0,sizeof(inst->auData));
        memset((char *)inst->sData,0,sizeof(inst->sData));
        memset((char *)inst->auDataBefore,0,sizeof(inst->auDataBefore));
        memset((char *)inst->sDataBefore,0,sizeof(inst->sDataBefore));

        inst->udCurrentAddr = inst->pWatchAddr + inst->iOffset;

        if (inst->pWatchAddr != 0 && (inst->udCurrentAddr > SHOW_LOCAL_PV_ADDR_SIZE))
        {
            memcpy((char *)inst->auData,(char *)inst->udCurrentAddr,sizeof(inst->auData));
            memcpy((char *)inst->sData,(char *)inst->udCurrentAddr,sizeof(inst->sData));
            memcpy((char *)inst->auDataBefore,(char *)inst->udCurrentAddr - SHOW_LOCAL_PV_ADDR_SIZE - 1,sizeof(inst->auDataBefore));
            memcpy((char *)inst->sDataBefore,(char *)inst->udCurrentAddr - SHOW_LOCAL_PV_ADDR_SIZE - 1,sizeof(inst->sDataBefore));
        }else
        {
            inst->uStatus = 1;//访问得到的地址为0
        }
    }
}
```

#### FB_ShowLocalPvAddrData.c - 显示局部变量的地址范围内内存分配
```c
/*!
	* @file      FB_ShowLocalPvAddrData.c
	* @brief     调用此函数，可观察当前任务下局部变量地址附近的内存分布情况
	* @date      创建于：2021.03.12；最后修改日期：2021.03.12
	* @version   V 1.00.1
	* @author    YuanZhiyi
	* @copyright B&R
*/
/*! History
 *****************************************************************************
 *     2021.03.12    V1.00.1   YuanZhiyi
 *         (new)     初始版本
 ******************************************************************************
*/

#include <bur/plctypes.h>
#include <string.h>
#ifdef __cplusplus
	extern "C"
	{
#endif
	#include "LxVar.h"
#ifdef __cplusplus
	};
#endif

void FB_ShowLocalPvAddrData(struct FB_ShowLocalPvAddrData* inst)
{
	//保证此函数可在被连续调用重复使用。
	if (memcmp((char *)inst->sName,(char *)inst->sNameTmp,sizeof(inst->sName)) != 0)
	{
		memcpy((char *)inst->sNameTmp,(char *)inst->sName,sizeof(inst->sName));
		inst->udCheckCallCount = 0;
	}

	if (inst->udCheckCallCount < 1)
	{
		memset((char *)inst->usArrData,0,sizeof(inst->usArrData));
		memcpy((char *)inst->FB_GetLocalPvAddrStrY.sPvName,(char *)inst->sName,sizeof(inst->sName));
		FB_GetLocalPvAddr(&inst->FB_GetLocalPvAddrStrY);
		if (inst->FB_GetLocalPvAddrStrY.udAddr != 0)
		{
			memcpy((char *)inst->usArrData,(char *)inst->FB_GetLocalPvAddrStrY.udAddr,sizeof(inst->usArrData));
		}
		inst->udAddr = inst->FB_GetLocalPvAddrStrY.udAddr;
	}
}
```

#### Strcats.c - 基于strlcat实现的缓冲区溢出保护的strcat
```c
/*!
	* @file      Strcats.c
	* @brief     防止内存溢出的安全型strcat
	* @date      创建于：2021.03.12；最后修改日期：2021.03.12
	* @version   V 1.00.1
	* @author    YuanZhiyi
	* @copyright B&R
*/
/*! History
 *****************************************************************************
 *     2021.03.12    V1.00.1   YuanZhiyi
 *         (new)     初始版本
 ******************************************************************************
*/

#include <bur/plctypes.h>
#include <string.h>
#ifdef __cplusplus
	extern "C"
	{
#endif
	#include "LxVar.h"
#ifdef __cplusplus
	};
#endif
/* TODO: Add your comment here */
//e.g. in ST : strcatsY(ADR('abc'),SIZEOF('abcXXXXXXX'),ADR('efg'),SIZEOF('efg'))
unsigned long Strcats(unsigned long pDest, unsigned long udDestsz, unsigned long pSrc)
{
	unsigned long udStrsz = 0;
	if (pDest == 0 || udDestsz == 0 || pSrc == 0)
	{
		//WarnLogWriteY(7210,(UDINT)"strcatsY Input parameters Error");
		return 7210;//strcatsY Input parameters Error
	}

	udStrsz = strlcat((char *)pDest,(char *)pSrc,udDestsz);
	return udStrsz;
}
```

#### Strcpys.c - 基于strlcpy实现的缓冲区溢出保护的strcpy
```c
/*!
	* @file      Strcpys.c
	* @brief     防止内存溢出的安全型strcpy
	* @date      创建于：2021.03.12；最后修改日期：2021.03.12
	* @version   V 1.00.1
	* @author    YuanZhiyi
	* @copyright B&R
*/
/*! History
 *****************************************************************************
 *     2021.03.12    V1.00.1   YuanZhiyi
 *         (new)     初始版本
 ******************************************************************************
*/

#include <bur/plctypes.h>
#include <string.h>
#ifdef __cplusplus
	extern "C"
	{
#endif
	#include "LxVar.h"
#ifdef __cplusplus
	};
#endif
/* TODO: Add your comment here */
//e.g. in ST : strcpys(ADR('abc'),SIZEOF('abcXXXXXXX'),ADR('efg'),SIZEOF('efg'))
unsigned long Strcpys(unsigned long pDest, unsigned long udDestsz, unsigned long pSrc)
{
	unsigned long udStrsz = 0;
	if (pDest == 0 || udDestsz == 0 || pSrc == 0)
	{
		//WarnLogWriteY(7211,(UDINT)"strcpysY Input parameters Error");
		return 7211;//strcpysY Input parameters Error
	}

	udStrsz = strlcpy((char *)pDest,(char *)pSrc,udDestsz);
	return udStrsz;
}
```

#### Strlens.c - 带有最大长度限制的字符串长度统计函数
```c
/*!
	* @file      Strlens.c
	* @brief     防止内存溢出的安全型strlen
	* @date      创建于：2021.03.12；最后修改日期：2021.03.12
	* @version   V 1.00.1
	* @author    YuanZhiyi
	* @copyright B&R
*/
/*! History
 *****************************************************************************
 *     2021.03.12    V1.00.1   YuanZhiyi
 *         (new)     初始版本
 ******************************************************************************
*/

#include <bur/plctypes.h>
#ifdef __cplusplus
	extern "C"
	{
#endif
	#include "LxVar.h"
	#include <string.h>
#ifdef __cplusplus
	};
#endif
/* TODO: Add your comment here */
unsigned long Strlens(unsigned long pStr, unsigned long udMaxSize)
{
	unsigned long udStrsz = 0;
	//检查数据入口
	if (pStr == 0 || udMaxSize ==  0)
	{
		//WarnLogWriteY(7214,(UDINT *)&"strnlenY input parameter Error");
		return 7214;//strnlenY input parameter Error;
	}

	//strnlen操作
	udStrsz = strnlen((char *)pStr,udMaxSize);

	return udStrsz;
}
```

#### FB_Udint2Str.c - 将UDINT类型数据转换为STRING
```c
/*!
	* @file        FB_Udint2Str.c
	* @brief       调用此函数，可通过srtOut得到UDINT类型数据转换为字符串的信息，并能得到字符串的实际长度。
	* @date        创建于：2019.08.13；最后修改日期：2019.08.13
	* @version     V 1.00.1
	* @author      YuanZhiyi
	* @copyright   B&R
*/
/*! History
 *****************************************************************************
 *     2019.08.13    V1.00.1   YuanZhiyi
 *         (new)     初始版本
 ******************************************************************************
*/

#include <bur/plctypes.h>
#ifdef __cplusplus
	extern "C"
	{
#endif
	#include "LxVar.h"
	#include <AsBrStr.h>
    #include <string.h>
#ifdef __cplusplus
	};
#endif

void FB_Udint2Str(struct FB_Udint2Str* inst)
{
	memset((UDINT *)inst->strOut,0,sizeof(inst->strOut));
	if (inst->udInput > 2147483647LL && inst->udInput < 3000000000LL )
	{
		inst->uiLen = brsitoa((DINT)(inst->udInput - 1000000000LL), (UDINT)&inst->strOut);
		memcpy((UDINT *)inst->strOut,(UDINT *)"2",1);
	}else if (inst->udInput >= 3000000000LL && inst->udInput < 4000000000LL )
	{
		inst->uiLen = brsitoa((DINT)(inst->udInput - 2000000000LL), (UDINT) inst->strOut);
		memcpy((UDINT *)inst->strOut,(UDINT *)"3",1);
	}else if (inst->udInput >= 4000000000LL)
	{
		inst->uiLen = brsitoa((DINT)(inst->udInput - 3000000000LL), (UDINT) inst->strOut);
		memcpy((UDINT *)inst->strOut,(UDINT *)"4",1);
	}else{
		inst->uiLen = brsitoa((DINT)(inst->udInput), (UDINT) inst->strOut);
	}
}
```

- FB_Real2Str.cc - 带有小数点限制的REAL数据转换 (not shown)

- FB_LReal2Str.cc - 带有小数点限制的LREAL数据转换 (not shown)

#### VarWarnLogWrite.c - 在System中写Logger函数
```c
/*!
* @file        VarWarnLogWrite.c
 * @brief      调用此函数，输入故障码（UINT类型），输入字符串信息，即可在Looger中的System中生成Logger记录。
 * @date       创建于：2019.08.13；最后修改日期：2020.11.04
 * @version    V1.00.1
 * @author     YuanZhiyi
 * @copyright  B&R
*/
/*! History
 *****************************************************************************
 *     2020.11.04    V1.00.1   YuanZhiyi
 *         (new)     初始版本
 ******************************************************************************
*/

#include <bur/plctypes.h>
#ifdef __cplusplus
	extern "C"
	{
#endif
#include "LxVar.h"
#include <sys_lib.h>
#ifdef __cplusplus
	};
#endif

unsigned short VarWarnLogWrite(UINT uNum,UDINT psErrorInfo)
{
    if (psErrorInfo == 0)
    {
        ERRxwarning(uNum, 0, (char *)"VarLogWrite Input psErrorInfo is NULL");
    }else
    {
        ERRxwarning(uNum, 0, (char *)psErrorInfo);
    }
    return 0;
}
```

#### VarServLogWrite.c - 在System中写Logger函数，PLC进入SERV
```c
/*!
* @file         LxVar/VarServLogWrite.c
  * @brief      调用此函数，输入故障码（UINT类型），输入字符串信息，即可在Looger中的System中生成Logger记录,PLC会直接进入SERV。
  * @date       创建于：2021.03.18；最后修改日期：2021.03.18
  * @version    V1.00.1
  * @author     YuanZhiyi
  * @copyright  B&R
*/
/*! History
 *****************************************************************************
 *     2021.03.18    V1.00.1   YuanZhiyi
 *         (new)     初始版本
 ******************************************************************************
*/

#include <bur/plctypes.h>
#ifdef __cplusplus
	extern "C"
	{
#endif
	#include "LxVar.h"
    #include <sys_lib.h>
#ifdef __cplusplus
	};
#endif

plcbit VarServLogWrite(unsigned short uErrorNum, unsigned long psErrorInfo)
{
    if (psErrorInfo == 0)
    {
        ERRxwarning(uErrorNum, 0, (char *)"VarLogWrite Input psErrorInfo is NULL");
    }else
    {
        ERRxfatal(uErrorNum, 0, (char *)psErrorInfo);
    }
    return 0;
}
```

- FB_Dec2Hex.cc - 十进制数据转换为十六进制字符串数据 (not shown)

- FB_Hex2Dec.cc - 十六进制字符串数据转换为十进制数据 (not shown)

#### FB_GetPvEntireName.c - 输入变量，判断是否为基本数据类型，如果不是，则返回下一级信息
```c
/*!
	* @file        FB_GetPvEntireName.c
	* @brief       调用此函数，可获得变量的完整名称，并反馈剩余的资源
	* @date        创建于：2021.03.15；最后修改日期：2021.03.16
	* @version     V 1.00.1
	* @author      YuanZhiyi
	* @copyright   B&R
*/
/*! History
 *****************************************************************************
 *     2021.03.16    V1.00.1   YuanZhiyi
 *         (new)     初始版本
 ******************************************************************************
*/

#include <bur/plctypes.h>
#include <string.h>
#ifdef __cplusplus
	extern "C"
	{
#endif
	#include "LxVar.h"
#ifdef __cplusplus
	};
#endif

void FB_GetPvEntireName(struct FB_GetPvEntireName* inst)
{
    //判断是否变量名有变化 任务名与变量名作为输入源
    if ((memcmp((char *)inst->sName,(char *)inst->sNameTmp,sizeof(inst->sName)) != 0) ||
        (memcmp((char *)inst->sModuleName,(char *)inst->sModuleNameTmp,sizeof(inst->sModuleName)) != 0)) {
        memcpy((char *)inst->sNameTmp,(char *)inst->sName,sizeof(inst->sName));
        memcpy((char *)inst->sModuleNameTmp,(char *)inst->sModuleName,sizeof(inst->sModuleName));

        inst->uCurrentIndex = 0;
        inst->uTotalNumber = 0;
        inst->bInTraversal = 0;
        inst->uStatus = 0;
        inst->bEnd = 0;
        memset((char *)inst->sEntirePvName,0,sizeof(inst->sEntirePvName));
        memset((char *)inst->sCompleteName,0,sizeof(inst->sCompleteName));
        memset((char *)inst->sCompleteNameTmp,0,sizeof(inst->sCompleteNameTmp));
    }

    //判断整体变量名是否有变化，
    if (memcmp((char *)inst->sCompleteName,(char *)inst->sCompleteNameTmp,sizeof(inst->sCompleteNameTmp)) != 0) {
	    memcpy((char *)inst->sCompleteNameTmp,(char *)inst->sCompleteName,sizeof(inst->sCompleteName));

        inst->uCurrentIndex = 0;
        inst->uTotalNumber = 0;
        inst->bInTraversal = 0;
        inst->uStatus = 0;
        inst->bEnd = 0;
        memset((char *)inst->sEntirePvName,0,sizeof(inst->sEntirePvName));
        memset((char *)inst->sModuleName,0,sizeof(inst->sModuleName));
        memset((char *)inst->sModuleNameTmp,0,sizeof(inst->sModuleNameTmp));
        memset((char *)inst->sName,0,sizeof(inst->sName));
        memset((char *)inst->sNameTmp,0,sizeof(inst->sNameTmp));
    }

    if (inst->bInTraversal == 0) { //仅在有变化时读取信息,此处默认为第一次对变量进行遍历
        //读取变量名信息
        if (memcmp((char *)inst->sCompleteName,(char *)"",1) != 0) {
            memcpy((char *)inst->FB_GetPvInfo_0.sCompleteName,(char *)inst->sCompleteName,sizeof(inst->sCompleteName));
        }else {
            memcpy((char *)inst->FB_GetPvInfo_0.sAppModuleName,(char *)inst->sModuleName,sizeof(inst->sModuleName));
            memcpy((char *)inst->FB_GetPvInfo_0.sName,(char *)inst->sName,sizeof(inst->sName));
        }
        inst->uTotalNumber = 0;
        inst->uCurrentIndex = 0;
        FB_GetPvInfo(&inst->FB_GetPvInfo_0); //异常情况判断
        if ((inst->FB_GetPvInfo_0.status != 0) && (inst->FB_GetPvInfo_0.status != 7001)) {
            inst->uStatus = inst->FB_GetPvInfo_0.status;
            return;
        }else { //拼接数据判断
            if (inst->FB_GetPvInfo_0.uDataType == 0 || inst->FB_GetPvInfo_0.uDataType == 15 ) {
                if (memcmp((char *)inst->sCompleteName,(char *)"",1) != 0) {
                    memcpy((char *)inst->FB_GetStruPvMemName_0.sCompleteName,(char *)inst->sCompleteName,sizeof(inst->sCompleteName));
                }else {
                    memcpy((char *)inst->FB_GetStruPvMemName_0.sModuleName,(char *)inst->sModuleName,sizeof(inst->sModuleName));
                    memcpy((char *)inst->FB_GetStruPvMemName_0.sName,(char *)inst->sName,sizeof(inst->sName));
                }
                FB_GetStruPvMemName(&inst->FB_GetStruPvMemName_0);
                if (inst->FB_GetStruPvMemName_0.uiStatus != 0) {
                    inst->uStatus = inst->FB_GetStruPvMemName_0.uiStatus;
                    return;
                }else {
                    memcpy((char *)inst->sEntirePvName,(char *)inst->FB_GetPvInfo_0.sPvName,sizeof(inst->FB_GetPvInfo_0.sPvName));
                    Strcats((UDINT)inst->sEntirePvName,sizeof(inst->sEntirePvName),(UDINT)".");
                    Strcats((UDINT)inst->sEntirePvName,sizeof(inst->sEntirePvName),(UDINT)inst->FB_GetStruPvMemName_0.sArrMemName[inst->uCurrentIndex]);
                    inst->uTotalNumber = inst->FB_GetStruPvMemName_0.uiMemNum;
                    if (inst->uCurrentIndex < inst->uTotalNumber) {
                        inst->uCurrentIndex++;
                    }
                    if (inst->FB_GetStruPvMemName_0.uiMemNum > 1)
                    {
                        inst->uStatus = 65535;
                        inst->bInTraversal = 1;
                    }
                }
            }else if(inst->FB_GetPvInfo_0.uiDimension > 1) {
                inst->uTotalNumber = inst->FB_GetPvInfo_0.uiDimension;
                memcpy((char *)inst->sEntirePvName,(char *)inst->FB_GetPvInfo_0.sPvName,sizeof(inst->FB_GetPvInfo_0.sPvName));
                Strcats((UDINT)inst->sEntirePvName,sizeof(inst->sEntirePvName),(UDINT)"[");
                inst->FB_Udint2Str_0.udInput = inst->uCurrentIndex;
                FB_Udint2Str(&inst->FB_Udint2Str_0);
                Strcats((UDINT)inst->sEntirePvName,sizeof(inst->sEntirePvName),(UDINT)inst->FB_Udint2Str_0.strOut);
                Strcats((UDINT)inst->sEntirePvName,sizeof(inst->sEntirePvName),(UDINT)"]");
                if (inst->uCurrentIndex < inst->uTotalNumber) {
                    inst->uCurrentIndex++;
                }
                inst->uStatus = 65535;
                inst->bInTraversal = 1;
            }else {
                memcpy((char *)inst->sEntirePvName,(char *)inst->FB_GetPvInfo_0.sPvName,sizeof(inst->FB_GetPvInfo_0.sPvName));
                inst->bEnd = 1;
            }
        }
        //当在遍历过程中
    } else if (inst->uCurrentIndex != 0 && inst->uTotalNumber != 0 && inst->bInTraversal == 1) {
        if ((inst->FB_GetPvInfo_0.uDataType == 0) || (inst->FB_GetPvInfo_0.uDataType == 15)) { //对结构信息的处理
            memcpy((char *)inst->sEntirePvName,(char *)inst->FB_GetPvInfo_0.sPvName,sizeof(inst->FB_GetPvInfo_0.sPvName));
            Strcats((UDINT)inst->sEntirePvName,sizeof(inst->sEntirePvName),(UDINT)".");
            Strcats((UDINT)inst->sEntirePvName,sizeof(inst->sEntirePvName),(UDINT)inst->FB_GetStruPvMemName_0.sArrMemName[inst->uCurrentIndex]);
            if (inst->uCurrentIndex < inst->uTotalNumber) {
                inst->uCurrentIndex++;
            }
            if (inst->uCurrentIndex >= inst->uTotalNumber) {
                inst->bInTraversal = 0;
                inst->uStatus = 0;
            }
        }else { //对数组类型数据进行处理
            memcpy((char *)inst->sEntirePvName,(char *)inst->FB_GetPvInfo_0.sPvName,sizeof(inst->FB_GetPvInfo_0.sPvName));
            Strcats((UDINT)inst->sEntirePvName,sizeof(inst->sEntirePvName),(UDINT)"[");
            inst->FB_Udint2Str_0.udInput = inst->uCurrentIndex;
            FB_Udint2Str(&inst->FB_Udint2Str_0);
            Strcats((UDINT)inst->sEntirePvName,sizeof(inst->sEntirePvName),(UDINT)inst->FB_Udint2Str_0.strOut);
            Strcats((UDINT)inst->sEntirePvName,sizeof(inst->sEntirePvName),(UDINT)"]");
            if (inst->uCurrentIndex < inst->uTotalNumber) {
                inst->uCurrentIndex++;
            }
            if (inst->uCurrentIndex >= inst->uTotalNumber) {
                inst->bInTraversal = 0;
                inst->uStatus = 0;
            }
        }
    }
}
```

#### ReturnPvAddr.c - 可获得变量地址信息，如果找不到，则进入SERV
```c
/*!
	* @file       LxVar/ReturnPvAddr.c
	* @brief      调用此函数，可获得变量地址信息，如果找不到，则进入SERV。
	* @date       创建于：2021.03.18；最后修改日期：2021.03.18
	* @version    V 1.00.1
	* @author     YuanZhiyi
	* @copyright  B&R
*/
/*! History
 *****************************************************************************
 *     2021.03.18    V1.00.1   YuanZhiyi
 *         (new)     初始版本
 ******************************************************************************
*/
/*! USE CASE

    .Var文件中申明变量为Reference变量
    *************************************
    VAR
    	Test0 : REFERENCE TO UDINT;
    END_VAR
    *************************************

    在.st代码中通过以下写法实现访问任意变量
    *************************************
    Test0 ACCESS ReturnPvAddr(ADR('gTest0'));
    *************************************

    如果变量找不到，则PLC进入SERV，并在Logger中记录找不到的变量名

 */

#include <bur/plctypes.h>
#include <sys_lib.h>
#include <string.h>
#ifdef __cplusplus
	extern "C"
	{
#endif
	#include "LxVar.h"
#ifdef __cplusplus
	};
#endif

unsigned long ReturnPvAddr(unsigned long psVarName)
{
    UDINT uPvAddr;
    UDINT uLength;
    STRING sErrorMsg[160];

    PV_xgetadr((char *)psVarName, (UDINT *)&uPvAddr, (UDINT *)&uLength);

    if (uPvAddr == 0) {
        memset((char *)sErrorMsg,0,sizeof(sErrorMsg));
        Strcpys((UDINT)sErrorMsg,sizeof(sErrorMsg),(UDINT)psVarName);
        Strcats((UDINT)sErrorMsg,sizeof(sErrorMsg),(UDINT)" Not Found");
        VarServLogWrite(55520,(UDINT)sErrorMsg);
    }
    return uPvAddr;
}
```

#### FB_ContinualStrcat.c - 可具有保护的,用于连续strcat操作的函数,避免负载过高
```c
/*!
	* @file      FB_ContinualStrcat.c
	* @brief     可具有保护的,用于连续strcat操作的函数,避免负载过高
	* @date      创建于：2021.06.03；
	* @author    YuanZhiyi
	* @copyright B&R
*/
/*! History
 *****************************************************************************
 *     2021.06.03    V1.00.1   YuanZhiyi
 *         (new)     初始版本
 *     2021.06.09    V1.00.2   YuanZhiyi
 *         (new)     增加uStrSize，整体字符串长度输出接口
 *     2022.10.31    V1.00.3   YuanZhiyi
 *         (new)     增加可选的uDestStrOffset，从目标字符串的某一偏移量开始进行字符串添加
 ******************************************************************************
*/
/*! Attention
 *****************************************************************************
    inst->uSrcMaxSize与inst->uDestMaxSize均为可选项，若不输入，则不进行安全检查
    此函数的目的为替换strcat函数，避免当字符串较大时，Strcat在找Dest的地址消耗过多资源
 ******************************************************************************
*/

#include <bur/plctypes.h>
#ifdef __cplusplus
	extern "C"
	{
#endif
	#include "LxVar.h"
    #include <string.h>
#ifdef __cplusplus
	};
#endif

void FB_ContinualStrcat(struct FB_ContinualStrcat* inst)
{
    if (inst->bInitial == 1) {
        inst->uOffset = 0;
        inst->bInitial = 0;
        if (inst->uDestMaxSize == 0) {
            /*----------在没有输入uDestMaxSize的情况下的执行方式---------------*/
            inst->uOffset = strlen((char *)inst->psDestStr + inst->uDestStrOffset) + inst->uDestStrOffset;
        }
        else {
            inst->uOffset = Strlens(inst->psDestStr + inst->uDestStrOffset,inst->uDestMaxSize) + inst->uDestStrOffset;
        }
    }

    if (inst->psSrcStr == 0 || inst->psDestStr == 0) {
        inst->uStatus = 7210; //输入地址为NULL
    }
    else {
        if (inst->uSrcMaxSize == 0) {
            /*----------在没有输入uSrcMax的情况下的执行方式---------------*/
            inst->uSrcActualLenth = strlen((char *)inst->psSrcStr);
        }
        else {
            inst->uSrcActualLenth = Strlens(inst->psSrcStr,inst->uSrcMaxSize);
        }

        /*-----------------进行目标地址边界检查，若没有输入uDestMaxSize，则不判断---------------*/
        if (inst->uOffset + inst->uSrcActualLenth > inst->uDestMaxSize && inst->uDestMaxSize != 0) {
            inst->uStatus = 7211; //超出目标地址最大长度。
        }
        else {
            memcpy((char *)(inst->psDestStr + inst->uOffset),(char *)inst->psSrcStr,inst->uSrcActualLenth);
            inst->uOffset = inst->uOffset + inst->uSrcActualLenth;
        }
    }

    /*----------------- 输出字符串整体长度---------------*/
    inst->uStrSize = inst->uOffset;
}
```

### Library Logical/Libraries/BrRand (ANSIC, version 1.00.4) - Random Value Generate
Depends on: sys_lib

#### BrRand.fun - 随机数生成库
```iecst
FUNCTION RandomBase : DINT (*随机数基础函数*)
END_FUNCTION

FUNCTION RandRange : DINT (*随机数范围函数*) (*$GROUP=User,$CAT=User,$GROUPICON=User.png,$CATICON=User.png*)
	VAR_INPUT
		min : DINT;
		max : DINT;
	END_VAR
END_FUNCTION

FUNCTION RandBOOL : BOOL (*输出BOOL随机数*) (*$GROUP=User,$CAT=User,$GROUPICON=User.png,$CATICON=User.png*)
END_FUNCTION

FUNCTION RandUSINT : USINT (*输出USINT随机数*) (*$GROUP=User,$CAT=User,$GROUPICON=User.png,$CATICON=User.png*)
END_FUNCTION

FUNCTION RandSINT : SINT (*输出SINT随机数*) (*$GROUP=User,$CAT=User,$GROUPICON=User.png,$CATICON=User.png*)
END_FUNCTION

FUNCTION RandUINT : UINT (*输出UINT随机数*) (*$GROUP=User,$CAT=User,$GROUPICON=User.png,$CATICON=User.png*)
END_FUNCTION

FUNCTION RandINT : INT (*输出INT随机数*) (*$GROUP=User,$CAT=User,$GROUPICON=User.png,$CATICON=User.png*)
END_FUNCTION

FUNCTION RandUDINT : UDINT (*输出UDINT随机数*) (*$GROUP=User,$CAT=User,$GROUPICON=User.png,$CATICON=User.png*)
END_FUNCTION

FUNCTION RandDINT : DINT (*输出DINT随机数*) (*$GROUP=User,$CAT=User,$GROUPICON=User.png,$CATICON=User.png*)
END_FUNCTION

FUNCTION RandREAL : REAL (*输出REAL随机数*) (*$GROUP=User,$CAT=User,$GROUPICON=User.png,$CATICON=User.png*)
END_FUNCTION

FUNCTION RandLREAL : LREAL (*输出LREAL随机数*) (*$GROUP=User,$CAT=User,$GROUPICON=User.png,$CATICON=User.png*)
END_FUNCTION

FUNCTION RandRangeUnsigned : UDINT (*设定范围产生无符号整型随机数*) (*$GROUP=User,$CAT=User,$GROUPICON=User.png,$CATICON=User.png*)
	VAR_INPUT
		min : UDINT;
		max : UDINT;
	END_VAR
END_FUNCTION

FUNCTION RandRangeSigned : DINT (*设定范围产生有符号整型随机数*) (*$GROUP=User,$CAT=User,$GROUPICON=User.png,$CATICON=User.png*)
	VAR_INPUT
		min : DINT;
		max : DINT;
	END_VAR
END_FUNCTION

FUNCTION RandRangeReal : REAL (*设定范围产生浮点类型随机数*) (*$GROUP=User,$CAT=User,$GROUPICON=User.png,$CATICON=User.png*)
	VAR_INPUT
		min : REAL;
		max : REAL;
	END_VAR
END_FUNCTION

{REDUND_ERROR} {REDUND_UNREPLICABLE} FUNCTION_BLOCK FB_RandString (*生成随机字符串*) (*$GROUP=User,$CAT=User,$GROUPICON=User.png,$CATICON=User.png*)
	VAR_INPUT
		pString : {REDUND_UNREPLICABLE} UDINT; (*[Optional]生成随机字符串地址*)
		uStrLen : {REDUND_UNREPLICABLE} UDINT; (*[Optional]设定的生成随机字符串长度，若为0则充满pString*)
	END_VAR
	VAR_OUTPUT
		sStrOut : {REDUND_UNREPLICABLE} STRING[8]; (*默认输出8个字节的随机字符串*)
	END_VAR
END_FUNCTION_BLOCK
```

#### RandomBase.c - 随机数基础函数
```c
/*!
* @file        BrRand/RandomBase.c
* @brief       调用此函数，实现DINT类型的随机数生成
* @date        创建于：2018.01.16 最后修改日期：2021.02.07
* @version     V 1.00.1
* @author      YuanZhiyi
* @copyright   B&R
*/
/*! History
 *****************************************************************************
 *     2021.02.07    V1.00.1   YuanZhiyi
 *         (new)     完成版本
 ******************************************************************************
*/
/*! Descripiton
 *****************************************************************************
 *
 ******************************************************************************
*/

#include <bur/plctypes.h>
#include <stdlib.h>
#ifdef __cplusplus
	extern "C"
	{
#endif
#include "BrRand.h"
#ifdef __cplusplus
	};
#endif

int rand();

signed long RandomBase(void)
{
    signed long i = 0;
    if ( rand()  > 1073741823 ) {
        i =  rand();
    }else {
        i = -1 * rand();
    }
    return i;
}
```

#### RandRange.c - 随机数范围函数
```c
/*!
* @file        BrRand/RandRange.c
* @brief       调用此函数，可实现随机数范围设置
* @date        创建于：2018.01.16 最后修改日期：2021.02.07
* @version     V 1.00.1
* @author      YuanZhiyi
* @copyright   B&R
*/
/*! History
 *****************************************************************************
 *     2021.02.07    V1.00.1   YuanZhiyi
 *         (new)     完成版本
 ******************************************************************************
*/
/*! Descripiton
 *****************************************************************************
 *
 ******************************************************************************
*/

#include <bur/plctypes.h>
#include <stdlib.h>
#ifdef __cplusplus
	extern "C"
	{
#endif
	#include "BrRand.h"
#ifdef __cplusplus
	};
#endif

int rand();

DINT RandRange(DINT min, DINT max)
{
	if (min > max) {
		return 0;
	} else if ((min == 0) && (max == 0)) {
		return RandomBase();
	} else if(min == max){
		return min;
    }else {
        // Note -  This will bias the randomness slightly, but probably not anything to be concerned about if you're not doing something particularly sensitive.
        return rand() % (max + 1 - min) + min;
    }
}
```

#### RandBOOL.c - 输出BOOL随机数
```c
/*!
* @file        BrRand/RandBOOL.c
* @brief       调用此函数，可实现BOOL类型数据随机生成
* @date        创建于：2018.01.16 最后修改日期：2021.02.07
* @version     V 1.00.1
* @author      YuanZhiyi
* @copyright   B&R
*/
/*! History
 *****************************************************************************
 *     2021.02.07    V1.00.1   YuanZhiyi
 *         (new)     完成版本
 ******************************************************************************
*/
/*! Descripiton
 *****************************************************************************
 *     使用案例: PV := RandBOOL();
 ******************************************************************************
*/

#include <bur/plctypes.h>
#include <stdlib.h>
#ifdef __cplusplus
	extern "C"
	{
#endif
	#include "BrRand.h"
#ifdef __cplusplus
	};
#endif

extern int rand();

plcbit RandBOOL(void)
{
	if (RandomBase() > 0) {
		return 1;
	} else {
		return 0;
	}
}
```

#### RandUSINT.c - 输出USINT随机数
```c
/*!
* @file        BrRand/RandUSINT.c
* @brief       调用此函数，可实现USINT类型数据随机生成
* @date        创建于：2018.01.16 最后修改日期：2021.02.07
* @version     V 1.00.1
* @author      YuanZhiyi
* @copyright   B&R
*/
/*! History
 *****************************************************************************
 *     2021.02.07    V1.00.1   YuanZhiyi
 *         (new)     完成版本
 ******************************************************************************
*/
/*! Descripiton
 *****************************************************************************
 *     使用案例: PV := RandUSINT();
 ******************************************************************************
*/

#include <bur/plctypes.h>
#include <stdlib.h>
#ifdef __cplusplus
	extern "C"
	{
#endif
	#include "BrRand.h"
#ifdef __cplusplus
	};
#endif

unsigned char RandUSINT()
{
	return abs(RandRange(0,0)) % 255;
}
```

#### RandSINT.c - 输出SINT随机数
```c
/*!
* @file        BrRand/RandSINT.c
* @brief       调用此函数，可实现SINT类型数据随机生成
* @date        创建于：2018.01.16 最后修改日期：2021.02.07
* @version     V 1.00.1
* @author      YuanZhiyi
* @copyright   B&R
*/
/*! History
 *****************************************************************************
 *     2021.02.07    V1.00.1   YuanZhiyi
 *         (new)     完成版本
 ******************************************************************************
*/
/*! Descripiton
 *****************************************************************************
 *     使用案例: PV := RandSINT();
 ******************************************************************************
*/

#include <bur/plctypes.h>
#include <stdlib.h>
#ifdef __cplusplus
	extern "C"
	{
#endif
#include "BrRand.h"
#ifdef __cplusplus
	};
#endif

signed char RandSINT()
{
    signed char tmpValue;
    tmpValue = RandRange(0,0) % 128;
    return tmpValue;
}
```

#### RandUINT.c - 输出UINT随机数
```c
/*!
* @file        BrRand/RandUINT.c
* @brief       调用此函数，可实现UINT类型数据随机生成
* @date        创建于：2018.01.16 最后修改日期：2021.02.07
* @version     V 1.00.1
* @author      YuanZhiyi
* @copyright   B&R
*/
/*! History
 *****************************************************************************
 *     2021.02.07    V1.00.1   YuanZhiyi
 *         (new)     完成版本
 ******************************************************************************
*/
/*! Descripiton
 *****************************************************************************
 *     使用案例: PV := RandUINT();
 ******************************************************************************
*/

#include <bur/plctypes.h>
#include <stdlib.h>
#ifdef __cplusplus
	extern "C"
	{
#endif
	#include "BrRand.h"
#ifdef __cplusplus
	};
#endif

unsigned short RandUINT()
{
	return abs(RandRange(0,0)) % 65535;
}
```

#### RandINT.c - 输出INT随机数
```c
/*!
* @file        BrRand/RandINT.c
* @brief       调用此函数，可实现INT类型数据随机生成
* @date        创建于：2018.01.16 最后修改日期：2021.02.07
* @version     V 1.00.1
* @author      YuanZhiyi
* @copyright   B&R
*/
/*! History
 *****************************************************************************
 *     2021.02.07    V1.00.1   YuanZhiyi
 *         (new)     完成版本
 ******************************************************************************
*/
/*! Descripiton
 *****************************************************************************
 *     使用案例: PV := RandINT();
 ******************************************************************************
*/

#include <bur/plctypes.h>
#include <stdlib.h>
#ifdef __cplusplus
	extern "C"
	{
#endif
	#include "BrRand.h"
#ifdef __cplusplus
	};
#endif

signed short RandINT()
{
    signed short tmpValue;
    tmpValue = RandRange(0,0) % 32768;
    return tmpValue;
}
```

#### RandUDINT.c - 输出UDINT随机数
```c
/*!
* @file        BrRand/RandUDINT.c
* @brief       调用此函数，可实现UDINT类型数据随机生成
* @date        创建于：2018.01.16 最后修改日期：2021.02.07
* @version     V 1.00.1
* @author      YuanZhiyi
* @copyright   B&R
*/
/*! History
 *****************************************************************************
 *     2021.02.07    V1.00.1   YuanZhiyi
 *         (new)     完成版本
 ******************************************************************************
*/
/*! Descripiton
 *****************************************************************************
 *     使用案例: PV := RandUDINT();
 ******************************************************************************
*/

#include <bur/plctypes.h>
#include <stdlib.h>
#ifdef __cplusplus
	extern "C"
	{
#endif
#include "BrRand.h"
#ifdef __cplusplus
	};
#endif

UDINT RandUDINT()
{
    return abs(RandRange(0,0)) * 2 + RandRange(0,1) ;
}
```

#### RandDINT.c - 输出DINT随机数
```c
/*!
* @file        BrRand/RandDINT.c
* @brief       调用此函数，可实现DINT类型数据随机生成
* @date        创建于：2018.01.16 最后修改日期：2021.02.07
* @version     V 1.00.1
* @author      YuanZhiyi
* @copyright   B&R
*/
/*! History
 *****************************************************************************
 *     2021.02.07    V1.00.1   YuanZhiyi
 *         (new)     完成版本
 ******************************************************************************
*/
/*! Descripiton
 *****************************************************************************
 *     使用案例: PV := RandDINT();
 ******************************************************************************
*/

#include <bur/plctypes.h>
#include <stdlib.h>
#ifdef __cplusplus
	extern "C"
	{
#endif
	#include "BrRand.h"
#ifdef __cplusplus
	};
#endif

DINT RandDINT()
{
    DINT iTmpValue;
    iTmpValue = RandomBase();
    return iTmpValue;
}
```

#### RandREAL.c - 输出REAL随机数
```c
/*!
* @file        BrRand/RandREAL.c
* @brief       调用此函数，可实现REAL类型数据随机生成
* @date        创建于：2018.01.16 最后修改日期：2021.02.07
* @version     V 1.00.1
* @author      YuanZhiyi
* @copyright   B&R
*/
/*! History
 *****************************************************************************
 *     2021.02.07    V1.00.1   YuanZhiyi
 *         (new)     完成版本
 ******************************************************************************
*/
/*! Descripiton
 *****************************************************************************
 *     使用案例: PV := RandREAL();
 ******************************************************************************
*/

#include <bur/plctypes.h>
#include <stdlib.h>
#ifdef __cplusplus
	extern "C"
	{
#endif
	#include "BrRand.h"
#ifdef __cplusplus
	};
#endif

REAL RandREAL()
{
    REAL tmpValue;
    tmpValue = (float)RandomBase() * (float)RandomBase() * (float)RandomBase() / (float)RandRange(1,2147483647) * RandSINT();
    return tmpValue;
}
```

#### RandLREAL.c - 输出LREAL随机数
```c
/*!
* @file        BrRand/RandLREAL.c
* @brief       调用此函数，可实现LREAL类型数据随机生成
* @date        创建于：2018.01.16 最后修改日期：2021.02.07
* @version     V 1.00.1
* @author      YuanZhiyi
* @copyright   B&R
*/
/*! History
 *****************************************************************************
 *     2021.02.07    V1.00.1   YuanZhiyi
 *         (new)     完成版本
 ******************************************************************************
*/
/*! Descripiton
 *****************************************************************************
 *     使用案例: PV := RandLREAL();
 ******************************************************************************
*/

#include <bur/plctypes.h>
#include <stdlib.h>
#ifdef __cplusplus
	extern "C"
	{
#endif
	#include "BrRand.h"
#ifdef __cplusplus
	};
#endif

LREAL RandLREAL()
{
    LREAL tmpValue;
    tmpValue = RandREAL() * rand() * 3.14159 / RandRange(1,1000) * RandRange(0,0) * 2.19 * rand() *  RandSINT();
    if (rand() < 0) {
        tmpValue = tmpValue * -1.0;
    }
    return tmpValue;
}
```

#### RandRangeUnsigned.c - 设定范围产生无符号整型随机数
```c
/*!
* @file        BrRand/RandRangeUnsigned.c
* @brief       调用此函数，可实现指定范围的无符号整型数据随机生成
* @date        创建于：2018.01.16；最后修改日期：2021.05.16
* @version     V1.00.1
* @author      YuanZhiyi
* @copyright   B&R
*/
/*! History
 *****************************************************************************
 *     2021.05.16    V1.00.1   YuanZhiyi
 *         (new)     更新实现
 ******************************************************************************
*/
/*! Descripiton
 *****************************************************************************
 *     使用案例: PV := RandRangeUnsigned(5,200);
 ******************************************************************************
*/

#include <bur/plctypes.h>
#include <stdlib.h>
#ifdef __cplusplus
	extern "C"
	{
#endif
#include "BrRand.h"
#ifdef __cplusplus
	};
#endif

UDINT RandRangeUnsigned(UDINT min, UDINT max)
{
    if (min > 2147483647 && max > 2147483647) {
        return abs(RandRange(min - 2147483647,max - 2147483647)) + 2147483647;
    }else if (min <= 2147483647 && max > 2147483647 ) {
        if (rand() > 0 ){
            return RandRange(min,2147483647);
        }
        else{
            return RandRange(0,max - 2147483647) + 2147483647;
        }
    }else {
        return (abs(RandRange(min,max)) * 2 + RandRange(0,1)) / 2 ;
    }
}
```

#### RandRangeSigned.c - 设定范围产生有符号整型随机数
```c
/*!
* @file        BrRand/RandRangeSigned.c
* @brief       调用此函数，可实现指定范围的有符号整型数据随机生成
* @date        创建于：2018.01.16；最后修改日期：2021.02.07
* @version     V1.00.1
* @author      YuanZhiyi
* @copyright   B&R
*/
/*! History
 *****************************************************************************
 *     2021.02.07    V1.00.1   YuanZhiyi
 *         (new)     初步实现
 ******************************************************************************
*/
/*! Descripiton
 *****************************************************************************
 *     使用案例: PV := RandRangeSigned(-10,10);
 ******************************************************************************
*/

#include <bur/plctypes.h>
#ifdef __cplusplus
	extern "C"
	{
#endif
	#include "BrRand.h"
#ifdef __cplusplus
	};
#endif

DINT RandRangeSigned(DINT min, DINT max)
{
    return RandRange(min,max);
}
```

#### RandRangeReal.c - 设定范围产生浮点类型随机数
```c
/*!
* @file        BrRand/RandRangeReal.c
* @brief       调用此函数，可实现指定范围的有符号数据随机生成
* @date        创建于：2018.01.16 最后修改日期：2021.09.23
* @version     V 1.00.2
* @author      YuanZhiyi
* @copyright   B&R
*/
/*! History
 *****************************************************************************
 *     2018.01.16    V1.00.1   YuanZhiyi
 *         (new)     初始版本
 *     2021.09.23    V1.00.2   YuanZhiyi
 *         (fix)     修正当min，max数值为0~1范围内数值时，随机数输出异常的问题。
 ******************************************************************************
*/
/*! Descripiton
 *****************************************************************************
 *     使用案例: RandRangeReal(0.8,1);
 *     注意事项: 输入REAL类型数据范围为(-2147483,2147483)
 ******************************************************************************
*/

#include <bur/plctypes.h>
#ifdef __cplusplus
	extern "C"
	{
#endif
	#include "BrRand.h"
#ifdef __cplusplus
	};
#endif

REAL RandRangeReal(REAL min, REAL max)
{
    DINT tmpMin;
    DINT tmpMax;
    REAL tmpValue;
    tmpMin       = (DINT)(min * 1000);
    tmpMax       = (DINT)(max * 1000);
    tmpValue     = (REAL)RandRange(tmpMin,tmpMax);
    if (tmpValue < (REAL)tmpMin) {
        tmpValue = tmpValue + 1.0;
    }else if(tmpValue > (REAL)tmpMax) {
        tmpValue = tmpValue - 1.0;
    }
    return tmpValue / 1000.0;
}
```

#### FB_RandString.c - Sync生成随机字符串
```c
/*!
* @file        BrRand/FB_RandString.c
* @brief       调用此函数，可实现指定范围的字符串随机生成创建,同步函数
* @date        创建于：2018.01.16 最后修改日期：2021.02.07
* @version     V 1.00.1
* @author      YuanZhiyi
* @copyright   B&R
*/
/*! History
 *****************************************************************************
 *     2021.02.07    V1.00.1   YuanZhiyi
 *         (new)     完成版本
 ******************************************************************************
*/
/*! Descripiton
 *****************************************************************************
 *     使用用法:
            FB_RandString_0.pString  := ADR(sString);
            FB_RandString_0.uStrLen := SIZEOF(sString);
            FB_RandString_0();
 ******************************************************************************
*/

#include <bur/plctypes.h>
#include <stdlib.h>
#include <string.h>
#ifdef __cplusplus
	extern "C"
	{
#endif
	#include "BrRand.h"
#ifdef __cplusplus
	};
#endif

static char charset[] = "abcdefghijklmnopqrstuvwxyzABCDEFGHIJKLMNOPQRSTUVWXYZ0123456789,.-#'?!";

void FB_RandString(struct FB_RandString* inst)
{
    unsigned long uMaxStrNum = 0;
    int i = 0;

    if (inst->uStrLen < sizeof(inst->sStrOut) - 1){
        uMaxStrNum = sizeof(inst->sStrOut) - 1;
    }else{
        uMaxStrNum = inst->uStrLen - 1;
    }

    for (i = 0; i < uMaxStrNum; i++){
        int uKey = rand() % (int)(sizeof(charset) - 1);
        if (i < sizeof(inst->sStrOut) - 1) {
            if (inst->pString != 0 && inst->uStrLen != 0) {
                memcpy((char *)inst->pString + i,&charset[uKey],1);
            }
            memcpy(inst->sStrOut + i,&charset[uKey],1);
        }else{
            if (inst->pString != 0 && inst->uStrLen != 0) {
                memcpy((char *)inst->pString + i,&charset[uKey],1);
            }
        }
    }
    memset(inst->sStrOut + sizeof(inst->sStrOut),0,1);
    if (inst->pString != 0 && inst->uStrLen != 0) {
        memset((char *)inst->pString + uMaxStrNum,0,1);
    }
}
```

- Visualisation Logical/mappView (not shown)

- Project.language (not shown)

### Program Logical/Archive/DataGen (IEC)

#### Main.st
```iecst
PROGRAM _INIT
	(* Insert code here *)
	UtcDTGetTime_0.enable := TRUE;
	UtcDTGetTime_0();
	IF UtcDTGetTime_0.status = 0 THEN
		dtBtachStartTime := UtcDTGetTime_0.DT1;
		dtBtachEndTime := UtcDTGetTime_0.DT1;
	END_IF
	strBatchCode := 'SCP173';
	bBatchTriger := FALSE;
END_PROGRAM

PROGRAM _CYCLIC
	(* Insert code here *)
	strTimeStamp;
	strTimeStamp := DT_TO_STRING(dtTimeStamp);
	IP1 := RandINT();
	IP2 := RandINT();

	FP1 := RandRangeReal(0, 100);
	FP2 := RandRangeReal(0, 100);

	CV := RandRangeReal(0, 100);
	VPF := RandRangeReal(0, 100);
	WT := RandRangeReal(0, 100);

	F1 := RandRangeReal(0, 100);
	F2 := RandRangeReal(0, 100);
	F3 := RandRangeReal(0, 100);
	F4 := RandRangeReal(0, 100);
	F5 := RandRangeReal(0, 100);
	F6 := RandRangeReal(0, 100);
	F7 := RandRangeReal(0, 100);
	F8 := RandRangeReal(0, 100);
	F9 := RandRangeReal(0, 100);
	F10 := RandRangeReal(0, 100);
	F11 := RandRangeReal(0, 100);
	F12 := RandRangeReal(0, 100);
	F13 := RandRangeReal(0, 100);
	F14 := RandRangeReal(0, 100);
	F15 := RandRangeReal(0, 100);

	FP := RandRangeReal(0, 100);

	AP1 := RandRangeReal(0, 100);
	BP1 := RandRangeReal(0, 100);
	AP2 := RandRangeReal(0, 100);

	ST1 := RandRangeReal(0, 100);
	ST2 := RandRangeReal(0, 100);
	ST3 := RandRangeReal(0, 100);
	ST4 := RandRangeReal(0, 100);
	ST5 := RandRangeReal(0, 100);
	ST6 := RandRangeReal(0, 100);
	ST7 := RandRangeReal(0, 100);
	ST8 := RandRangeReal(0, 100);
	ST9 := RandRangeReal(0, 100);
	ST10 := RandRangeReal(0, 100);
	ST11 := RandRangeReal(0, 100);
	ST12 := RandRangeReal(0, 100);
	ST13 := RandRangeReal(0, 100);
	ST14 := RandRangeReal(0, 100);
	ST15 := RandRangeReal(0, 100);

	AIR := RandRangeReal(0, 100);
	CP := RandRangeReal(0, 100);
	CT := RandRangeReal(0, 100);
	CRT := RandRangeReal(0, 100);
	ES := RandRangeReal(0, 100);
	FT := RandRangeReal(0, 100);
	FF := RandRangeReal(0, 100);

	FC := RandINT();

	HT1 := RandRangeReal(0, 100);
	HT2 := RandRangeReal(0, 100);
	HT3 := RandRangeReal(0, 100);
	HT4 := RandRangeReal(0, 100);
	HT5 := RandRangeReal(0, 100);
	HT6 := RandRangeReal(0, 100);
	HT7 := RandRangeReal(0, 100);
	HT8 := RandRangeReal(0, 100);
	HT9 := RandRangeReal(0, 100);
	HT10 := RandRangeReal(0, 100);
	HT11 := RandRangeReal(0, 100);
	HT12 := RandRangeReal(0, 100);
	HT13 := RandRangeReal(0, 100);
	HT14 := RandRangeReal(0, 100);
	HT15 := RandRangeReal(0, 100);
	HT16 := RandRangeReal(0, 100);
	HT17 := RandRangeReal(0, 100);
	HT18 := RandRangeReal(0, 100);
	HT19 := RandRangeReal(0, 100);
	HT20 := RandRangeReal(0, 100);

	MP := RandRangeReal(0, 100);
	MT := RandRangeReal(0, 100);
	MCT := RandRangeReal(0, 100);
	MCP := RandRangeReal(0, 100);
	EC := RandRangeReal(0, 100);
	EST := RandRangeReal(0, 100);
	ES1 := RandRangeReal(0, 100);
	TC := RandRangeReal(0, 100);
	TF := RandRangeReal(0, 100);
	TW := RandRangeReal(0, 100);
END_PROGRAM

PROGRAM _EXIT
	(* Insert code here *)

END_PROGRAM
```

### Program Logical/Archive/DataRev (IEC)

#### Variables.var
```iecst
(*Insert your comment here.*)
VAR
	bExecuteRead : BOOL;
	stDbReadQuery : dbReadQuery_typ;
	bTestTriger : BOOL;
	uiHeartBeat : UINT;
	uiQueryFeedBack : UINT;
	udiStartTime : ARRAY[0..50] OF UDINT;
	udiEndTime : ARRAY[0..50] OF UDINT;
	strBatchCode : ARRAY[0..50] OF STRING[80];
	strStartTime : ARRAY[0..50] OF STRING[80];
	strEndTime : ARRAY[0..50] OF STRING[80];
	udiCursor : UDINT;
	diCursor : DINT;
	bNextPage : BOOL;
	bPrePage : BOOL;
	strBatchCode1 : STRING[80];
	strListName : ARRAY[0..50] OF STRING[80];
	bTriger : BOOL;
END_VAR
```

### Program Logical/Archive/AlarmQuerry (IEC) - 报警查询

#### Main.st - Init, cyclic, exit code
```iecst
PROGRAM _INIT
	(* Insert code here *)
	stDbReadQuery.stConfig.strPointName[0] := 'msg';
	guiDBHeartBeat;

END_PROGRAM

PROGRAM _CYCLIC
	(* Insert code here *)
	//Data GEN - Alarm Group 1 Data Points
	// GET TIME
	UtcDTGetTime_0.enable := TRUE;
	UtcDTGetTime_0();
	IF UtcDTGetTime_0.status = 0 THEN
		ts := DT_TO_STRING(UtcDTGetTime_0.DT1);
	END_IF

	Code := RandRange(1,10);  // 报警码
	msg := RandRange(1,10);  // 报警信息
	severity := RandRange(1,4);  // 报警等级 (1=Critical, 2=Major, 3=Minor, 4=Info)
	Status := btrigger;  // 报警状态 (TRUE=Active, FALSE=Cleared)
	Batch ;  // 生产批号

	//Triggerrecord
	btrigger;

	//Data from DATABASE
	bExecuteRead;
	stDbReadQuery;

	//Para and button connect
	stDbReadQuery.stConfig.strStartTime[0] := '';
	brsstrcat(ADR(stDbReadQuery.stConfig.strStartTime[0]),ADR(HMIAlarmQuerrystYear));
	brsstrcat(ADR(stDbReadQuery.stConfig.strStartTime[0]),ADR('-'));
	brsstrcat(ADR(stDbReadQuery.stConfig.strStartTime[0]),ADR(HMIAlarmQuerrystMonth));
	brsstrcat(ADR(stDbReadQuery.stConfig.strStartTime[0]),ADR('-'));
	brsstrcat(ADR(stDbReadQuery.stConfig.strStartTime[0]),ADR(HMIAlarmQuerrystDay));
	brsstrcat(ADR(stDbReadQuery.stConfig.strStartTime[0]),ADR(' '));

	brsstrcat(ADR(stDbReadQuery.stConfig.strStartTime[0]),ADR(HMIAlarmQuerrystHour));
	brsstrcat(ADR(stDbReadQuery.stConfig.strStartTime[0]),ADR(':'));
	brsstrcat(ADR(stDbReadQuery.stConfig.strStartTime[0]),ADR(HMIAlarmQuerrystMinute));
	brsstrcat(ADR(stDbReadQuery.stConfig.strStartTime[0]),ADR(':'));
	brsstrcat(ADR(stDbReadQuery.stConfig.strStartTime[0]),ADR(HMIAlarmQuerrystSec));

	stDbReadQuery.stConfig.strEndTime[0] := '';
	brsstrcat(ADR(stDbReadQuery.stConfig.strEndTime[0]),ADR(HMIAlarmQuerryedYear));
	brsstrcat(ADR(stDbReadQuery.stConfig.strEndTime[0]),ADR('-'));
	brsstrcat(ADR(stDbReadQuery.stConfig.strEndTime[0]),ADR(HMIAlarmQuerryedMonth));
	brsstrcat(ADR(stDbReadQuery.stConfig.strEndTime[0]),ADR('-'));
	brsstrcat(ADR(stDbReadQuery.stConfig.strEndTime[0]),ADR(HMIAlarmQuerryedDay));
	brsstrcat(ADR(stDbReadQuery.stConfig.strEndTime[0]),ADR(' '));

	brsstrcat(ADR(stDbReadQuery.stConfig.strEndTime[0]),ADR(HMIAlarmQuerryedHour));
	brsstrcat(ADR(stDbReadQuery.stConfig.strEndTime[0]),ADR(':'));
	brsstrcat(ADR(stDbReadQuery.stConfig.strEndTime[0]),ADR(HMIAlarmQuerryedMinute));
	brsstrcat(ADR(stDbReadQuery.stConfig.strEndTime[0]),ADR(':'));
	brsstrcat(ADR(stDbReadQuery.stConfig.strEndTime[0]),ADR(HMIAlarmQuerryedSec));

	bExecuteRead := UINT_TO_BOOL(HMIAlarmQuerryMBBtn);

	//Response data
	FOR i := 0 TO MAX_ENTRIES_PERPAGE_MINUSONE DO
		IF stDbReadQuery.stRev[0].udiRevTime[i] <> 0 THEN
			//强制转换
			DT_TO_DTStructure(UDINT_TO_DT(stDbReadQuery.stRev[0].udiRevTime[i]),ADR(stRecvDT[i]));

			HMIAlarmQuerryTimestr[i] := '';

			brsitoa(UINT_TO_DINT(stRecvDT[i].year),ADR(strempYear));
			brsitoa(UINT_TO_DINT(stRecvDT[i].month),ADR(strempMonth));
			brsitoa(UINT_TO_DINT(stRecvDT[i].day),ADR(strempDay));
			brsitoa(UINT_TO_DINT(stRecvDT[i].hour),ADR(strempHour));
			brsitoa(UINT_TO_DINT(stRecvDT[i].minute),ADR(strempMinute));
			brsitoa(UINT_TO_DINT(stRecvDT[i].second),ADR(strtempSecond));

			brsstrcat(ADR(HMIAlarmQuerryTimestr[i]),ADR(strempYear));
			brsstrcat(ADR(HMIAlarmQuerryTimestr[i]),ADR('-'));
			brsstrcat(ADR(HMIAlarmQuerryTimestr[i]),ADR(strempMonth));
			brsstrcat(ADR(HMIAlarmQuerryTimestr[i]),ADR('-'));
			brsstrcat(ADR(HMIAlarmQuerryTimestr[i]),ADR(strempDay));
			brsstrcat(ADR(HMIAlarmQuerryTimestr[i]),ADR(' '));
			brsstrcat(ADR(HMIAlarmQuerryTimestr[i]),ADR(strempHour));
			brsstrcat(ADR(HMIAlarmQuerryTimestr[i]),ADR(':'));
			brsstrcat(ADR(HMIAlarmQuerryTimestr[i]),ADR(strempMinute));
			brsstrcat(ADR(HMIAlarmQuerryTimestr[i]),ADR(':'));
			brsstrcat(ADR(HMIAlarmQuerryTimestr[i]),ADR(strtempSecond));

		ELSE
			brsmemset(ADR(HMIAlarmQuerryTimestr[i]),0,SIZEOF(HMIAlarmQuerryTimestr[i]));
		END_IF
		HMIAlarmQuerryIndex[i] :=  REAL_TO_UINT(stDbReadQuery.stRev[0].rRevBuffer[i]);

	END_FOR

	IF EDGEPOS(UINT_TO_BOOL(HMIAlarmClearMBBtn)) THEN
		brsmemset(ADR(stDbReadQuery.stRev), 0, SIZEOF(stDbReadQuery.stRev));
	END_IF

END_PROGRAM

PROGRAM _EXIT
	(* Insert code here *)

END_PROGRAM
```

#### Variables.var - Local variables
```iecst
(*HMIConnect*)
VAR
	HMIAlarmQuerrystYear : STRING[10];
	HMIAlarmQuerrystMonth : STRING[10];
	HMIAlarmQuerrystDay : STRING[10];
	HMIAlarmQuerrystHour : STRING[10];
	HMIAlarmQuerrystMinute : STRING[10];
	HMIAlarmQuerrystSec : STRING[10];
	HMIAlarmQuerryedYear : STRING[10];
	HMIAlarmQuerryedMonth : STRING[10];
	HMIAlarmQuerryedDay : STRING[10];
	HMIAlarmQuerryedHour : STRING[10];
	HMIAlarmQuerryedMinute : STRING[10];
	HMIAlarmQuerryedSec : STRING[10];
	HMIAlarmClearMBBtn : UINT;
	HMIAlarmQuerryMBBtn : UINT;
	HMIAlarmQuerryTimestr : ARRAY[0..MAX_ENTRIES_PERPAGE_MINUSONE] OF STRING[100];
	HMIAlarmQuerryIndex : ARRAY[0..MAX_ENTRIES_PERPAGE_MINUSONE] OF UINT;
END_VAR
(*DATA BASE Query*)
VAR
	bExecuteRead : BOOL;
	stDbReadQuery : dbReadQuery_typ;
END_VAR
(*Data point*)
VAR
	ts : STRING[80];
	Code : DINT;
	msg : DINT;
	Batch : DINT;
	severity : DINT;
	Status : DINT;
END_VAR
(*TIME CONVENT*)
VAR
	UtcDTGetTime_0 : UtcDTGetTime;
END_VAR
(*connect var*)
VAR
	stRecvDT : {REDUND_UNREPLICABLE} ARRAY[0..MAX_ENTRIES_PERPAGE_MINUSONE] OF DTStructure;
	strtempSecond : STRING[10];
	strempMinute : STRING[10];
	strempHour : STRING[10];
	strempDay : STRING[10];
	strempMonth : STRING[10];
	strempYear : STRING[10];
	i : UINT;
END_VAR
(*Insert your comment here.*)
VAR CONSTANT
	MAX_ENTRIES_PERPAGE_MINUSONE : UINT := MAX_ENTRIES_PERPAGE- 1;
	MAX_ENTRIES_PERPAGE : UINT := 15;
END_VAR
VAR
	btrigger : BOOL;
END_VAR
```

### Program Logical/Archive/Trend (IEC)

#### Variables.var
```iecst
(*DATA BASE Query*)
VAR
	stDbReadQuery : dbReadQuery_typ;
	bExecuteRead : BOOL;
END_VAR
(*DATA BASE CONSTANT*)
VAR CONSTANT
	REV_BUFFER_SIZE : UINT := 10000;
	REV_BUFFER_SIZE_MINUS_ONE : UINT := REV_BUFFER_SIZE-1;
	DB_READ_QUERY_SIZE : UINT := 10;
	DB_READ_QUERY_SIZE_MINUS_ONE : UINT := DB_READ_QUERY_SIZE-1;
END_VAR
(*Insert your comment here.*)
VAR CONSTANT
	MAX_ENTRIES_PERPAGE_MINUSONE : UINT := MAX_ENTRIES_PERPAGE- 1;
	MAX_ENTRIES_PERPAGE : UINT := 15;
END_VAR
VAR
	Trenddata : DINT;
END_VAR
```

#### Main.st
```iecst
PROGRAM _INIT
	(* Insert code here *)

END_PROGRAM

PROGRAM _CYCLIC
	(* Insert code here *)
		//Data GEN
	Trenddata:= RandRange(1,10);

	stDbReadQuery;
	bExecuteRead;

END_PROGRAM

PROGRAM _EXIT
	(* Insert code here *)

END_PROGRAM
```

### Program Logical/Archive/ParallelTest (IEC) - 并发触发测试

#### Variables.var
```iecst
VAR
	usiTestModel : USINT;
	usiIdx : USINT;
	rCollectorIntervalSeconds : REAL := 5.0;
END_VAR
(*Insert your comment here.*)
VAR
	bExecuteRead : BOOL;
	stDbReadQuery : dbReadQuery_typ;
	bParallelTriger : ARRAY[0..MY_DATA_SIZE_MINUS_ONE] OF BOOL;
	uiHeartBeat : UINT;
	uiQueryFeedBack : UINT;
END_VAR
(*DATA POINT*)
VAR
	F1 : ARRAY[0..MY_DATA_SIZE_MINUS_ONE] OF REAL;
	F2 : ARRAY[0..MY_DATA_SIZE_MINUS_ONE] OF REAL;
	F3 : ARRAY[0..MY_DATA_SIZE_MINUS_ONE] OF REAL;
	F4 : ARRAY[0..MY_DATA_SIZE_MINUS_ONE] OF REAL;
	F5 : ARRAY[0..MY_DATA_SIZE_MINUS_ONE] OF REAL;
END_VAR
(*CONSTANT*)
VAR CONSTANT
	MY_DATA_SIZE : UDINT := 100;
	MY_DATA_SIZE_MINUS_ONE : UDINT := MY_DATA_SIZE-1;
END_VAR
```
